LIN {X 0,Y 282.326,Z 515.053,A -85,B 0,C 180,E1 -18846.21,E2 -18846.21} C_VEL
LIN {X 0,Y 281.83,Z 513.099,A -85,B 0,C 180,E1 -18846.511,E2 -18846.511} C_VEL
LIN {X 0,Y 278.434,Z 504.389,A -85,B 0,C 180,E1 -18848.429,E2 -18848.429} C_VEL
LIN {X 0,Y 275.799,Z 498.647,A -85,B 0,C 180,E1 -18850.051,E2 -18850.051} C_VEL
LIN {X 0,Y 272.892,Z 492.622,A -85,B 0,C 180,E1 -18852.108,E2 -18852.108} C_VEL
LIN {X 0,Y 269.449,Z 485.759,A -85,B 0,C 180,E1 -18855.232,E2 -18855.232} C_VEL
LIN {X 0,Y 266.756,Z 480.992,A -85,B 0,C 180,E1 -18859.021,E2 -18859.021} C_VEL
LIN {X 0,Y 265.964,Z 478.887,A -85,B 0,C 180,E1 -18861.776,E2 -18861.776} C_VEL
LIN {X 0,Y 265.924,Z 478.099,A -85,B 0,C 180,E1 -18863.476,E2 -18863.476} C_VEL
LIN {X 0,Y 267.159,Z 478.377,A -85,B 0,C 180,E1 -18867.333,E2 -18867.333} C_VEL
LIN {X 0,Y 268.305,Z 478.984,A -85,B 0,C 180,E1 -18868.98,E2 -18868.98} C_VEL
LIN {X 0,Y 271.621,Z 482.626,A -85,B 0,C 180,E1 -18872.425,E2 -18872.425} C_VEL
LIN {X 0,Y 274.885,Z 486.681,A -85,B 0,C 180,E1 -18874.84,E2 -18874.84} C_VEL
LIN {X 0,Y 277.888,Z 490.776,A -85,B 0,C 180,E1 -18876.655,E2 -18876.655} C_VEL
LIN {X 0,Y 281.533,Z 496.331,A -85,B 0,C 180,E1 -18878.583,E2 -18878.583} C_VEL
LIN {X 0,Y 285.637,Z 503.762,A -85,B 0,C 180,E1 -18880.525,E2 -18880.525} C_VEL
LIN {X 0,Y 286.557,Z 505.613,A -85,B 0,C 180,E1 -18880.936,E2 -18880.936} C_VEL
LIN {X 0,Y 280.795,Z 557.104,A -85,B 0,C 180,E1 -18882.994,E2 -18882.994} C_VEL
LIN {X 0,Y 279.087,Z 570.067,A -85,B 0,C 180,E1 -18883.788,E2 -18883.788} C_VEL
LIN {X 0,Y 276.843,Z 582.59,A -85,B 0,C 180,E1 -18884.824,E2 -18884.824} C_VEL
LIN {X 0,Y 274.127,Z 594.365,A -85,B 0,C 180,E1 -18886.092,E2 -18886.092} C_VEL
LIN {X 0,Y 270.959,Z 605.812,A -85,B 0,C 180,E1 -18887.644,E2 -18887.644} C_VEL
LIN {X 0,Y 267.715,Z 616.024,A -85,B 0,C 180,E1 -18889.411,E2 -18889.411} C_VEL
LIN {X 0,Y 264.222,Z 625.564,A -85,B 0,C 180,E1 -18891.493,E2 -18891.493} C_VEL
LIN {X 0,Y 261.46,Z 632.41,A -85,B 0,C 180,E1 -18893.362,E2 -18893.362} C_VEL
LIN {X 0,Y 258.787,Z 638.353,A -85,B 0,C 180,E1 -18895.327,E2 -18895.327} C_VEL
LIN {X 0,Y 256.164,Z 643.857,A -85,B 0,C 180,E1 -18897.641,E2 -18897.641} C_VEL
LIN {X 0,Y 253.889,Z 648.134,A -85,B 0,C 180,E1 -18900,E2 -18900} C_VEL
LIN {X 0,Y 252.583,Z 650.359,A -85,B 0,C 180,E1 -18901.594,E2 -18901.594} C_VEL
LIN {X 0,Y 251.382,Z 652.245,A -85,B 0,C 180,E1 -18903.321,E2 -18903.321} C_VEL
LIN {X 0,Y 250.422,Z 653.517,A -85,B 0,C 180,E1 -18904.83,E2 -18904.83} C_VEL
LIN {X 0,Y 249.542,Z 654.406,A -85,B 0,C 180,E1 -18906.468,E2 -18906.468} C_VEL
LIN {X 0,Y 248.726,Z 654.929,A -85,B 0,C 180,E1 -18908.517,E2 -18908.517} C_VEL
LIN {X 0,Y 247.846,Z 654.521,A -85,B 0,C 180,E1 -18911.449,E2 -18911.449} C_VEL
LIN {X 0,Y 247.554,Z 653.658,A -85,B 0,C 180,E1 -18913.127,E2 -18913.127} C_VEL
LIN {X 0,Y 247.381,Z 652.208,A -85,B 0,C 180,E1 -18914.997,E2 -18914.997} C_VEL
LIN {X 0,Y 247.276,Z 649.517,A -85,B 0,C 180,E1 -18917.363,E2 -18917.363} C_VEL
LIN {X 0,Y 247.484,Z 645.518,A -85,B 0,C 180,E1 -18919.924,E2 -18919.924} C_VEL
LIN {X 0,Y 247.988,Z 639.143,A -85,B 0,C 180,E1 -18922.934,E2 -18922.934} C_VEL
LIN {X 0,Y 248.657,Z 632.173,A -85,B 0,C 180,E1 -18925.487,E2 -18925.487} C_VEL
LIN {X 0,Y 249.458,Z 624.632,A -85,B 0,C 180,E1 -18927.701,E2 -18927.701} C_VEL
LIN {X 0,Y 250.533,Z 614.804,A -85,B 0,C 180,E1 -18930.03,E2 -18930.03} C_VEL
LIN {X 0,Y 251.705,Z 604.3,A -85,B 0,C 180,E1 -18932.04,E2 -18932.04} C_VEL
LIN {X 0,Y 252.873,Z 593.019,A -85,B 0,C 180,E1 -18933.769,E2 -18933.769} C_VEL
LIN {X 0,Y 254.011,Z 580.659,A -85,B 0,C 180,E1 -18935.28,E2 -18935.28} C_VEL
LIN {X 0,Y 255.061,Z 566.615,A -85,B 0,C 180,E1 -18936.574,E2 -18936.574} C_VEL
LIN {X 0,Y 255.819,Z 553.718,A -85,B 0,C 180,E1 -18937.433,E2 -18937.433} C_VEL
LIN {X 0,Y 256.516,Z 534.013,A -85,B 0,C 180,E1 -18938.276,E2 -18938.276} C_VEL
LIN {X 0,Y 258.671,Z 480.462,A -85,B 0,C 180,E1 -18940.334,E2 -18940.334} C_VEL
LIN {X 0,Y 249.04,Z 452.464,A -85,B 0,C 180,E1 -18942.125,E2 -18942.125} C_VEL
LIN {X 0,Y 248.985,Z 452.468,A -85,B 0,C 180,E1 -18945.116,E2 -18945.116} C_VEL
LIN {X 0,Y 249.008,Z 452.464,A -85,B 0,C 180,E1 -18947.36,E2 -18947.36} C_VEL
LIN {X 0,Y 249.024,Z 452.466,A -85,B 0,C 180,E1 -18952.206,E2 -18952.206} C_VEL
LIN {X 0,Y 249.045,Z 452.459,A -85,B 0,C 180,E1 -18955.639,E2 -18955.639} C_VEL
LIN {X 0,Y 249.004,Z 452.465,A -85,B 0,C 180,E1 -18959.466,E2 -18959.466} C_VEL
LIN {X 0,Y 249.037,Z 452.46,A -85,B 0,C 180,E1 -18963.157,E2 -18963.157} C_VEL
LIN {X 0,Y 249.06,Z 452.461,A -85,B 0,C 180,E1 -18966.73,E2 -18966.73} C_VEL
LIN {X 0,Y 249.112,Z 452.454,A -85,B 0,C 180,E1 -18970.211,E2 -18970.211} C_VEL
LIN {X 0,Y 249.244,Z 452.435,A -85,B 0,C 180,E1 -18973.621,E2 -18973.621} C_VEL
LIN {X 0,Y 249.241,Z 452.438,A -85,B 0,C 180,E1 -18978.615,E2 -18978.615} C_VEL
LIN {X 0,Y 249.419,Z 452.413,A -85,B 0,C 180,E1 -18981.9,E2 -18981.9} C_VEL
LIN {X 0,Y 249.28,Z 452.432,A -85,B 0,C 180,E1 -18985.148,E2 -18985.148} C_VEL
LIN {X 0,Y 249.673,Z 452.385,A -85,B 0,C 180,E1 -18988.386,E2 -18988.386} C_VEL
LIN {X 0,Y 249.672,Z 452.382,A -85,B 0,C 180,E1 -18991.612,E2 -18991.612} C_VEL
LIN {X 0,Y 249.446,Z 452.413,A -85,B 0,C 180,E1 -18996.47,E2 -18996.47} C_VEL
LIN {X 0,Y 249.344,Z 452.422,A -85,B 0,C 180,E1 -18999.736,E2 -18999.736} C_VEL
LIN {X 0,Y 249.184,Z 452.445,A -85,B 0,C 180,E1 -19004.704,E2 -19004.704} C_VEL
LIN {X 0,Y 249.112,Z 452.452,A -85,B 0,C 180,E1 -19008.079,E2 -19008.079} C_VEL
LIN {X 0,Y 249.08,Z 452.456,A -85,B 0,C 180,E1 -19011.518,E2 -19011.518} C_VEL
LIN {X 0,Y 249.086,Z 452.453,A -85,B 0,C 180,E1 -19015.46,E2 -19015.46} C_VEL
LIN {X 0,Y 249.039,Z 452.463,A -85,B 0,C 180,E1 -19018.974,E2 -19018.974} C_VEL
LIN {X 0,Y 249.026,Z 452.466,A -85,B 0,C 180,E1 -19022.426,E2 -19022.426} C_VEL
LIN {X 0,Y 249.046,Z 452.462,A -85,B 0,C 180,E1 -19026.342,E2 -19026.342} C_VEL
LIN {X 0,Y 248.983,Z 452.472,A -85,B 0,C 180,E1 -19030.482,E2 -19030.482} C_VEL
LIN {X 0,Y 248.993,Z 452.468,A -85,B 0,C 180,E1 -19032.788,E2 -19032.788} C_VEL
LIN {X 0,Y 249.008,Z 452.465,A -85,B 0,C 180,E1 -19037.361,E2 -19037.361} C_VEL
LIN {X 0,Y 249.024,Z 452.46,A -85,B 0,C 180,E1 -19041.619,E2 -19041.619} C_VEL
LIN {X 0,Y 249.042,Z 452.461,A -85,B 0,C 180,E1 -19045.639,E2 -19045.639} C_VEL
LIN {X 0,Y 249.046,Z 452.458,A -85,B 0,C 180,E1 -19049.472,E2 -19049.472} C_VEL
LIN {X 0,Y 249.071,Z 452.458,A -85,B 0,C 180,E1 -19053.162,E2 -19053.162} C_VEL
LIN {X 0,Y 249.079,Z 452.458,A -85,B 0,C 180,E1 -19056.733,E2 -19056.733} C_VEL
LIN {X 0,Y 249.11,Z 452.452,A -85,B 0,C 180,E1 -19060.212,E2 -19060.212} C_VEL
LIN {X 0,Y 249.241,Z 452.436,A -85,B 0,C 180,E1 -19063.622,E2 -19063.622} C_VEL
LIN {X 0,Y 249.252,Z 452.436,A -85,B 0,C 180,E1 -19068.617,E2 -19068.617} C_VEL
LIN {X 0,Y 249.477,Z 452.407,A -85,B 0,C 180,E1 -19071.903,E2 -19071.903} C_VEL
LIN {X 0,Y 249.433,Z 452.414,A -85,B 0,C 180,E1 -19076.77,E2 -19076.77} C_VEL
LIN {X 0,Y 249.727,Z 452.376,A -85,B 0,C 180,E1 -19080,E2 -19080} C_VEL
LIN {X 0,Y 249.435,Z 452.411,A -85,B 0,C 180,E1 -19083.231,E2 -19083.231} C_VEL
LIN {X 0,Y 249.484,Z 452.406,A -85,B 0,C 180,E1 -19088.097,E2 -19088.097} C_VEL
LIN {X 0,Y 249.253,Z 452.434,A -85,B 0,C 180,E1 -19091.384,E2 -19091.384} C_VEL
LIN {X 0,Y 249.241,Z 452.437,A -85,B 0,C 180,E1 -19096.378,E2 -19096.378} C_VEL
LIN {X 0,Y 249.083,Z 452.454,A -85,B 0,C 180,E1 -19101.519,E2 -19101.519} C_VEL
LIN {X 0,Y 249.117,Z 452.452,A -85,B 0,C 180,E1 -19105.476,E2 -19105.476} C_VEL
LIN {X 0,Y 249.083,Z 452.457,A -85,B 0,C 180,E1 -19108.994,E2 -19108.994} C_VEL
LIN {X 0,Y 249.03,Z 452.462,A -85,B 0,C 180,E1 -19112.426,E2 -19112.426} C_VEL
LIN {X 0,Y 249.039,Z 452.462,A -85,B 0,C 180,E1 -19114.761,E2 -19114.761} C_VEL
LIN {X 0,Y 248.388,Z 452.546,A -85,B 0,C 180,E1 -19116.111,E2 -19116.111} C_VEL
LIN {X 0,Y 245.555,Z 452.903,A -85,B 0,C 180,E1 -19118.312,E2 -19118.312} C_VEL
LIN {X 0,Y 243.118,Z 453.205,A -85,B 0,C 180,E1 -19120.104,E2 -19120.104} C_VEL
LIN {X 0,Y 242.04,Z 453.334,A -85,B 0,C 180,E1 -19121.494,E2 -19121.494} C_VEL
LIN {X 0,Y 241.936,Z 453.345,A -85,B 0,C 180,E1 -19121.966,E2 -19121.966} C_VEL
LIN {X 0,Y 241.936,Z 453.349,A -85,B 0,C 180,E1 -19126.571,E2 -19126.571} C_VEL
LIN {X 0,Y 241.956,Z 453.343,A -85,B 0,C 180,E1 -19130.282,E2 -19130.282} C_VEL
LIN {X 0,Y 242.063,Z 453.369,A -85,B 0,C 180,E1 -19133.471,E2 -19133.471} C_VEL
LIN {X 0,Y 244.715,Z 466.337,A -85,B 0,C 180,E1 -19137.907,E2 -19137.907} C_VEL
LIN {X 0,Y 246.665,Z 475.875,A -85,B 0,C 180,E1 -19141.03,E2 -19141.03} C_VEL
LIN {X 0,Y 246.306,Z 479.6,A -85,B 0,C 180,E1 -19142.144,E2 -19142.144} C_VEL
LIN {X 0,Y 248.483,Z 510.094,A -85,B 0,C 180,E1 -19143.6,E2 -19143.6} C_VEL
LIN {X 0,Y 250.829,Z 535.634,A -85,B 0,C 180,E1 -19144.809,E2 -19144.809} C_VEL
LIN {X 0,Y 248.607,Z 589.384,A -85,B 0,C 180,E1 -19147.017,E2 -19147.017} C_VEL
LIN {X 0,Y 247.623,Z 603.29,A -85,B 0,C 180,E1 -19147.911,E2 -19147.911} C_VEL
LIN {X 0,Y 246.363,Z 616.413,A -85,B 0,C 180,E1 -19149.11,E2 -19149.11} C_VEL
LIN {X 0,Y 245.144,Z 628.254,A -85,B 0,C 180,E1 -19150.533,E2 -19150.533} C_VEL
LIN {X 0,Y 243.955,Z 638.928,A -85,B 0,C 180,E1 -19152.149,E2 -19152.149} C_VEL
LIN {X 0,Y 242.763,Z 648.961,A -85,B 0,C 180,E1 -19154.037,E2 -19154.037} C_VEL
LIN {X 0,Y 241.855,Z 658.034,A -85,B 0,C 180,E1 -19156.13,E2 -19156.13} C_VEL
LIN {X 0,Y 241.155,Z 665.499,A -85,B 0,C 180,E1 -19158.23,E2 -19158.23} C_VEL
LIN {X 0,Y 240.709,Z 672.776,A -85,B 0,C 180,E1 -19160.76,E2 -19160.76} C_VEL
LIN {X 0,Y 240.581,Z 678.564,A -85,B 0,C 180,E1 -19163.332,E2 -19163.332} C_VEL
LIN {X 0,Y 240.581,Z 682.853,A -85,B 0,C 180,E1 -19165.812,E2 -19165.812} C_VEL
LIN {X 0,Y 240.687,Z 686.021,A -85,B 0,C 180,E1 -19168.327,E2 -19168.327} C_VEL
LIN {X 0,Y 240.697,Z 687.509,A -85,B 0,C 180,E1 -19170.001,E2 -19170.001} C_VEL
LIN {X 0,Y 240.551,Z 688.525,A -85,B 0,C 180,E1 -19171.675,E2 -19171.675} C_VEL
LIN {X 0,Y 240.183,Z 689.037,A -85,B 0,C 180,E1 -19173.356,E2 -19173.356} C_VEL
LIN {X 0,Y 240.093,Z 689.117,A -85,B 0,C 180,E1 -19175.586,E2 -19175.586} C_VEL
LIN {X 0,Y 240.16,Z 688.153,A -85,B 0,C 180,E1 -19178.414,E2 -19178.414} C_VEL
LIN {X 0,Y 240.473,Z 687.031,A -85,B 0,C 180,E1 -19180.1,E2 -19180.1} C_VEL
LIN {X 0,Y 241.585,Z 683.542,A -85,B 0,C 180,E1 -19183.458,E2 -19183.458} C_VEL
LIN {X 0,Y 243.176,Z 679.816,A -85,B 0,C 180,E1 -19185.936,E2 -19185.936} C_VEL
LIN {X 0,Y 245.077,Z 675.065,A -85,B 0,C 180,E1 -19188.388,E2 -19188.388} C_VEL
LIN {X 0,Y 248.042,Z 668.056,A -85,B 0,C 180,E1 -19191.178,E2 -19191.178} C_VEL
LIN {X 0,Y 251.761,Z 659.198,A -85,B 0,C 180,E1 -19193.878,E2 -19193.878} C_VEL
LIN {X 0,Y 255.594,Z 649.847,A -85,B 0,C 180,E1 -19196.101,E2 -19196.101} C_VEL
LIN {X 0,Y 259.509,Z 639.305,A -85,B 0,C 180,E1 -19198.071,E2 -19198.071} C_VEL
LIN {X 0,Y 263.479,Z 627.709,A -85,B 0,C 180,E1 -19199.789,E2 -19199.789} C_VEL
LIN {X 0,Y 267.052,Z 616.215,A -85,B 0,C 180,E1 -19201.097,E2 -19201.097} C_VEL
LIN {X 0,Y 270.567,Z 602.674,A -85,B 0,C 180,E1 -19202.284,E2 -19202.284} C_VEL
LIN {X 0,Y 273.295,Z 589,A -85,B 0,C 180,E1 -19203.18,E2 -19203.18} C_VEL
LIN {X 0,Y 275.538,Z 574.021,A -85,B 0,C 180,E1 -19203.86,E2 -19203.86} C_VEL
LIN {X 0,Y 279.213,Z 541.099,A -85,B 0,C 180,E1 -19205.196,E2 -19205.196} C_VEL
LIN {X 0,Y 279.022,Z 528.795,A -85,B 0,C 180,E1 -19206.177,E2 -19206.177} C_VEL
LIN {X 0,Y 278.4,Z 518.134,A -85,B 0,C 180,E1 -19207.26,E2 -19207.26} C_VEL
LIN {X 0,Y 275.283,Z 509.663,A -85,B 0,C 180,E1 -19209.169,E2 -19209.169} C_VEL
LIN {X 0,Y 272.972,Z 504.355,A -85,B 0,C 180,E1 -19210.707,E2 -19210.707} C_VEL
LIN {X 0,Y 270.596,Z 498.97,A -85,B 0,C 180,E1 -19212.564,E2 -19212.564} C_VEL
LIN {X 0,Y 267.41,Z 492.248,A -85,B 0,C 180,E1 -19215.677,E2 -19215.677} C_VEL
LIN {X 0,Y 265.082,Z 487.715,A -85,B 0,C 180,E1 -19219.345,E2 -19219.345} C_VEL
LIN {X 0,Y 264.402,Z 485.554,A -85,B 0,C 180,E1 -19222.312,E2 -19222.312} C_VEL
LIN {X 0,Y 264.526,Z 484.953,A -85,B 0,C 180,E1 -19224.232,E2 -19224.232} C_VEL
LIN {X 0,Y 266.105,Z 485.466,A -85,B 0,C 180,E1 -19228.115,E2 -19228.115} C_VEL
LIN {X 0,Y 266.971,Z 486.316,A -85,B 0,C 180,E1 -19229.286,E2 -19229.286} C_VEL
LIN {X 0,Y 269.719,Z 489.366,A -85,B 0,C 180,E1 -19232.161,E2 -19232.161} C_VEL
LIN {X 0,Y 272.655,Z 493.167,A -85,B 0,C 180,E1 -19234.446,E2 -19234.446} C_VEL
LIN {X 0,Y 275.309,Z 497.029,A -85,B 0,C 180,E1 -19236.173,E2 -19236.173} C_VEL
LIN {X 0,Y 278.098,Z 501.457,A -85,B 0,C 180,E1 -19237.779,E2 -19237.779} C_VEL
LIN {X 0,Y 281.912,Z 508.483,A -85,B 0,C 180,E1 -19239.743,E2 -19239.743} C_VEL
LIN {X 0,Y 282.164,Z 509.341,A -85,B 0,C 180,E1 -19239.89,E2 -19239.89} C_VEL
LIN {X 0,Y 276.44,Z 557.647,A -85,B 0,C 180,E1 -19241.843,E2 -19241.843} C_VEL
LIN {X 0,Y 274.71,Z 570.009,A -85,B 0,C 180,E1 -19242.61,E2 -19242.61} C_VEL
LIN {X 0,Y 272.153,Z 583.297,A -85,B 0,C 180,E1 -19243.709,E2 -19243.709} C_VEL
LIN {X 0,Y 269.12,Z 595.783,A -85,B 0,C 180,E1 -19245.074,E2 -19245.074} C_VEL
LIN {X 0,Y 265.798,Z 606.936,A -85,B 0,C 180,E1 -19246.623,E2 -19246.623} C_VEL
LIN {X 0,Y 262.351,Z 616.95,A -85,B 0,C 180,E1 -19248.409,E2 -19248.409} C_VEL
LIN {X 0,Y 258.505,Z 626.84,A -85,B 0,C 180,E1 -19250.612,E2 -19250.612} C_VEL
LIN {X 0,Y 255.264,Z 634.243,A -85,B 0,C 180,E1 -19252.723,E2 -19252.723} C_VEL
LIN {X 0,Y 251.834,Z 641.075,A -85,B 0,C 180,E1 -19255.197,E2 -19255.197} C_VEL
LIN {X 0,Y 249.126,Z 646.135,A -85,B 0,C 180,E1 -19257.575,E2 -19257.575} C_VEL
LIN {X 0,Y 246.789,Z 650.03,A -85,B 0,C 180,E1 -19260,E2 -19260} C_VEL
LIN {X 0,Y 245.477,Z 652.035,A -85,B 0,C 180,E1 -19261.64,E2 -19261.64} C_VEL
LIN {X 0,Y 244.309,Z 653.549,A -85,B 0,C 180,E1 -19263.298,E2 -19263.298} C_VEL
LIN {X 0,Y 243.262,Z 654.657,A -85,B 0,C 180,E1 -19264.972,E2 -19264.972} C_VEL
LIN {X 0,Y 242.391,Z 655.359,A -85,B 0,C 180,E1 -19266.66,E2 -19266.66} C_VEL
LIN {X 0,Y 241.641,Z 655.588,A -85,B 0,C 180,E1 -19268.551,E2 -19268.551} C_VEL
LIN {X 0,Y 240.696,Z 654.78,A -85,B 0,C 180,E1 -19271.794,E2 -19271.794} C_VEL
LIN {X 0,Y 240.436,Z 653.716,A -85,B 0,C 180,E1 -19273.523,E2 -19273.523} C_VEL
LIN {X 0,Y 240.233,Z 651.242,A -85,B 0,C 180,E1 -19276.136,E2 -19276.136} C_VEL
LIN {X 0,Y 240.279,Z 647.625,A -85,B 0,C 180,E1 -19278.768,E2 -19278.768} C_VEL
LIN {X 0,Y 240.591,Z 642.722,A -85,B 0,C 180,E1 -19281.431,E2 -19281.431} C_VEL
LIN {X 0,Y 241.136,Z 636.448,A -85,B 0,C 180,E1 -19284.081,E2 -19284.081} C_VEL
LIN {X 0,Y 241.975,Z 628.435,A -85,B 0,C 180,E1 -19286.756,E2 -19286.756} C_VEL
LIN {X 0,Y 242.889,Z 620.108,A -85,B 0,C 180,E1 -19288.99,E2 -19288.99} C_VEL
LIN {X 0,Y 244.039,Z 609.913,A -85,B 0,C 180,E1 -19291.223,E2 -19291.223} C_VEL
LIN {X 0,Y 245.209,Z 598.821,A -85,B 0,C 180,E1 -19293.167,E2 -19293.167} C_VEL
LIN {X 0,Y 246.406,Z 587.366,A -85,B 0,C 180,E1 -19294.781,E2 -19294.781} C_VEL
LIN {X 0,Y 247.459,Z 575.374,A -85,B 0,C 180,E1 -19296.108,E2 -19296.108} C_VEL
LIN {X 0,Y 248.529,Z 560.848,A -85,B 0,C 180,E1 -19297.308,E2 -19297.308} C_VEL
LIN {X 0,Y 249.158,Z 547.242,A -85,B 0,C 180,E1 -19298.074,E2 -19298.074} C_VEL
LIN {X 0,Y 251.767,Z 481.763,A -85,B 0,C 180,E1 -19300.686,E2 -19300.686} C_VEL
LIN {X 0,Y 241.975,Z 453.345,A -85,B 0,C 180,E1 -19302.592,E2 -19302.592} C_VEL
LIN {X 0,Y 241.924,Z 453.35,A -85,B 0,C 180,E1 -19306.574,E2 -19306.574} C_VEL
LIN {X 0,Y 241.938,Z 453.349,A -85,B 0,C 180,E1 -19310.276,E2 -19310.276} C_VEL
LIN {X 0,Y 241.975,Z 453.343,A -85,B 0,C 180,E1 -19314.486,E2 -19314.486} C_VEL
LIN {X 0,Y 241.955,Z 453.348,A -85,B 0,C 180,E1 -19318.476,E2 -19318.476} C_VEL
LIN {X 0,Y 241.97,Z 453.344,A -85,B 0,C 180,E1 -19322.307,E2 -19322.307} C_VEL
LIN {X 0,Y 242.029,Z 453.336,A -85,B 0,C 180,E1 -19326.012,E2 -19326.012} C_VEL
LIN {X 0,Y 242.039,Z 453.333,A -85,B 0,C 180,E1 -19329.607,E2 -19329.607} C_VEL
LIN {X 0,Y 242.165,Z 453.317,A -85,B 0,C 180,E1 -19333.278,E2 -19333.278} C_VEL
LIN {X 0,Y 242.178,Z 453.319,A -85,B 0,C 180,E1 -19338.279,E2 -19338.279} C_VEL
LIN {X 0,Y 242.373,Z 453.29,A -85,B 0,C 180,E1 -19341.663,E2 -19341.663} C_VEL
LIN {X 0,Y 242.24,Z 453.309,A -85,B 0,C 180,E1 -19345.006,E2 -19345.006} C_VEL
LIN {X 0,Y 242.634,Z 453.261,A -85,B 0,C 180,E1 -19348.34,E2 -19348.34} C_VEL
LIN {X 0,Y 242.632,Z 453.259,A -85,B 0,C 180,E1 -19351.659,E2 -19351.659} C_VEL
LIN {X 0,Y 242.417,Z 453.287,A -85,B 0,C 180,E1 -19356.659,E2 -19356.659} C_VEL
LIN {X 0,Y 242.268,Z 453.305,A -85,B 0,C 180,E1 -19360.023,E2 -19360.023} C_VEL
LIN {X 0,Y 242.14,Z 453.319,A -85,B 0,C 180,E1 -19365.142,E2 -19365.142} C_VEL
LIN {X 0,Y 242.05,Z 453.335,A -85,B 0,C 180,E1 -19368.625,E2 -19368.625} C_VEL
LIN {X 0,Y 242.003,Z 453.34,A -85,B 0,C 180,E1 -19372.18,E2 -19372.18} C_VEL
LIN {X 0,Y 242.032,Z 453.332,A -85,B 0,C 180,E1 -19375.82,E2 -19375.82} C_VEL
LIN {X 0,Y 241.969,Z 453.342,A -85,B 0,C 180,E1 -19379.588,E2 -19379.588} C_VEL
LIN {X 0,Y 241.978,Z 453.338,A -85,B 0,C 180,E1 -19383.492,E2 -19383.492} C_VEL
LIN {X 0,Y 241.986,Z 453.34,A -85,B 0,C 180,E1 -19387.582,E2 -19387.582} C_VEL
LIN {X 0,Y 241.922,Z 453.347,A -85,B 0,C 180,E1 -19391.925,E2 -19391.925} C_VEL
LIN {X 0,Y 241.924,Z 453.352,A -85,B 0,C 180,E1 -19396.573,E2 -19396.573} C_VEL
LIN {X 0,Y 241.955,Z 453.345,A -85,B 0,C 180,E1 -19400.281,E2 -19400.281} C_VEL
LIN {X 0,Y 241.98,Z 453.344,A -85,B 0,C 180,E1 -19404.488,E2 -19404.488} C_VEL
LIN {X 0,Y 241.972,Z 453.345,A -85,B 0,C 180,E1 -19408.48,E2 -19408.48} C_VEL
LIN {X 0,Y 242.002,Z 453.339,A -85,B 0,C 180,E1 -19412.312,E2 -19412.312} C_VEL
LIN {X 0,Y 242.057,Z 453.332,A -85,B 0,C 180,E1 -19416.016,E2 -19416.016} C_VEL
LIN {X 0,Y 242.037,Z 453.331,A -85,B 0,C 180,E1 -19419.608,E2 -19419.608} C_VEL
LIN {X 0,Y 242.162,Z 453.318,A -85,B 0,C 180,E1 -19423.278,E2 -19423.278} C_VEL
LIN {X 0,Y 242.186,Z 453.314,A -85,B 0,C 180,E1 -19428.28,E2 -19428.28} C_VEL
LIN {X 0,Y 242.424,Z 453.285,A -85,B 0,C 180,E1 -19431.666,E2 -19431.666} C_VEL
LIN {X 0,Y 242.254,Z 453.306,A -85,B 0,C 180,E1 -19435.007,E2 -19435.007} C_VEL
LIN {X 0,Y 242.635,Z 453.26,A -85,B 0,C 180,E1 -19438.34,E2 -19438.34} C_VEL
LIN {X 0,Y 242.635,Z 453.259,A -85,B 0,C 180,E1 -19441.66,E2 -19441.66} C_VEL
LIN {X 0,Y 242.433,Z 453.286,A -85,B 0,C 180,E1 -19446.659,E2 -19446.659} C_VEL
LIN {X 0,Y 242.345,Z 453.296,A -85,B 0,C 180,E1 -19450.021,E2 -19450.021} C_VEL
LIN {X 0,Y 242.166,Z 453.318,A -85,B 0,C 180,E1 -19455.141,E2 -19455.141} C_VEL
LIN {X 0,Y 242.072,Z 453.333,A -85,B 0,C 180,E1 -19458.624,E2 -19458.624} C_VEL
LIN {X 0,Y 242.006,Z 453.336,A -85,B 0,C 180,E1 -19462.181,E2 -19462.181} C_VEL
LIN {X 0,Y 242.066,Z 453.33,A -85,B 0,C 180,E1 -19465.838,E2 -19465.838} C_VEL
LIN {X 0,Y 242.03,Z 453.333,A -85,B 0,C 180,E1 -19469.58,E2 -19469.58} C_VEL
LIN {X 0,Y 241.98,Z 453.34,A -85,B 0,C 180,E1 -19473.493,E2 -19473.493} C_VEL
LIN {X 0,Y 241.989,Z 453.339,A -85,B 0,C 180,E1 -19477.582,E2 -19477.582} C_VEL
LIN {X 0,Y 241.936,Z 453.345,A -85,B 0,C 180,E1 -19481.966,E2 -19481.966} C_VEL
LIN {X 0,Y 241.227,Z 453.436,A -85,B 0,C 180,E1 -19483.355,E2 -19483.355} C_VEL
LIN {X 0,Y 238.377,Z 453.789,A -85,B 0,C 180,E1 -19485.622,E2 -19485.622} C_VEL
LIN {X 0,Y 235.981,Z 454.09,A -85,B 0,C 180,E1 -19487.469,E2 -19487.469} C_VEL
LIN {X 0,Y 234.952,Z 454.217,A -85,B 0,C 180,E1 -19488.902,E2 -19488.902} C_VEL
LIN {X 0,Y 234.866,Z 454.224,A -85,B 0,C 180,E1 -19489.387,E2 -19489.387} C_VEL
LIN {X 0,Y 235.021,Z 454.306,A -85,B 0,C 180,E1 -19493.202,E2 -19493.202} C_VEL
LIN {X 0,Y 237.71,Z 467.519,A -85,B 0,C 180,E1 -19497.848,E2 -19497.848} C_VEL
LIN {X 0,Y 239.623,Z 476.982,A -85,B 0,C 180,E1 -19501.031,E2 -19501.031} C_VEL
LIN {X 0,Y 239.401,Z 478.938,A -85,B 0,C 180,E1 -19501.65,E2 -19501.65} C_VEL
LIN {X 0,Y 241.445,Z 508.632,A -85,B 0,C 180,E1 -19503.126,E2 -19503.126} C_VEL
LIN {X 0,Y 243.914,Z 535.614,A -85,B 0,C 180,E1 -19504.45,E2 -19504.45} C_VEL
LIN {X 0,Y 241.564,Z 589.707,A -85,B 0,C 180,E1 -19506.761,E2 -19506.761} C_VEL
LIN {X 0,Y 240.599,Z 603.374,A -85,B 0,C 180,E1 -19507.683,E2 -19507.683} C_VEL
LIN {X 0,Y 239.331,Z 616.305,A -85,B 0,C 180,E1 -19508.917,E2 -19508.917} C_VEL
LIN {X 0,Y 238.099,Z 628.024,A -85,B 0,C 180,E1 -19510.382,E2 -19510.382} C_VEL
LIN {X 0,Y 236.817,Z 639.25,A -85,B 0,C 180,E1 -19512.165,E2 -19512.165} C_VEL
LIN {X 0,Y 235.693,Z 648.551,A -85,B 0,C 180,E1 -19513.99,E2 -19513.99} C_VEL
LIN {X 0,Y 234.767,Z 657.567,A -85,B 0,C 180,E1 -19516.144,E2 -19516.144} C_VEL
LIN {X 0,Y 234.078,Z 664.993,A -85,B 0,C 180,E1 -19518.308,E2 -19518.308} C_VEL
LIN {X 0,Y 233.65,Z 672.236,A -85,B 0,C 180,E1 -19520.915,E2 -19520.915} C_VEL
LIN {X 0,Y 233.519,Z 677.516,A -85,B 0,C 180,E1 -19523.302,E2 -19523.302} C_VEL
LIN {X 0,Y 233.551,Z 681.673,A -85,B 0,C 180,E1 -19525.686,E2 -19525.686} C_VEL
LIN {X 0,Y 233.639,Z 685.012,A -85,B 0,C 180,E1 -19528.277,E2 -19528.277} C_VEL
LIN {X 0,Y 233.661,Z 686.583,A -85,B 0,C 180,E1 -19530.001,E2 -19530.001} C_VEL
LIN {X 0,Y 233.487,Z 687.681,A -85,B 0,C 180,E1 -19531.726,E2 -19531.726} C_VEL
LIN {X 0,Y 233.109,Z 688.311,A -85,B 0,C 180,E1 -19533.458,E2 -19533.458} C_VEL
LIN {X 0,Y 233.03,Z 688.498,A -85,B 0,C 180,E1 -19535.582,E2 -19535.582} C_VEL
LIN {X 0,Y 233.101,Z 687.69,A -85,B 0,C 180,E1 -19538.671,E2 -19538.671} C_VEL
LIN {X 0,Y 233.448,Z 686.687,A -85,B 0,C 180,E1 -19540.407,E2 -19540.407} C_VEL
LIN {X 0,Y 233.913,Z 685.281,A -85,B 0,C 180,E1 -19542.142,E2 -19542.142} C_VEL
LIN {X 0,Y 235.2,Z 682.394,A -85,B 0,C 180,E1 -19544.714,E2 -19544.714} C_VEL
LIN {X 0,Y 236.922,Z 678.523,A -85,B 0,C 180,E1 -19547.256,E2 -19547.256} C_VEL
LIN {X 0,Y 239.729,Z 672.449,A -85,B 0,C 180,E1 -19550.26,E2 -19550.26} C_VEL
LIN {X 0,Y 243.075,Z 665.266,A -85,B 0,C 180,E1 -19552.975,E2 -19552.975} C_VEL
LIN {X 0,Y 246.648,Z 657.384,A -85,B 0,C 180,E1 -19555.304,E2 -19555.304} C_VEL
LIN {X 0,Y 250.781,Z 647.803,A -85,B 0,C 180,E1 -19557.543,E2 -19557.543} C_VEL
LIN {X 0,Y 254.987,Z 637.136,A -85,B 0,C 180,E1 -19559.517,E2 -19559.517} C_VEL
LIN {X 0,Y 258.839,Z 626.51,A -85,B 0,C 180,E1 -19561.058,E2 -19561.058} C_VEL
LIN {X 0,Y 262.608,Z 614.873,A -85,B 0,C 180,E1 -19562.361,E2 -19562.361} C_VEL
LIN {X 0,Y 266.302,Z 601.416,A -85,B 0,C 180,E1 -19563.544,E2 -19563.544} C_VEL
LIN {X 0,Y 269.043,Z 588.511,A -85,B 0,C 180,E1 -19564.396,E2 -19564.396} C_VEL
LIN {X 0,Y 271.392,Z 573.761,A -85,B 0,C 180,E1 -19565.074,E2 -19565.074} C_VEL
LIN {X 0,Y 275.078,Z 542.504,A -85,B 0,C 180,E1 -19566.353,E2 -19566.353} C_VEL
LIN {X 0,Y 275.116,Z 531.447,A -85,B 0,C 180,E1 -19567.272,E2 -19567.272} C_VEL
LIN {X 0,Y 274.738,Z 522.333,A -85,B 0,C 180,E1 -19568.2,E2 -19568.2} C_VEL
LIN {X 0,Y 272.158,Z 514.807,A -85,B 0,C 180,E1 -19569.983,E2 -19569.983} C_VEL
LIN {X 0,Y 270.216,Z 510.059,A -85,B 0,C 180,E1 -19571.4,E2 -19571.4} C_VEL
LIN {X 0,Y 268.024,Z 504.852,A -85,B 0,C 180,E1 -19573.252,E2 -19573.252} C_VEL
LIN {X 0,Y 265.419,Z 498.75,A -85,B 0,C 180,E1 -19576.138,E2 -19576.138} C_VEL
LIN {X 0,Y 263.452,Z 494.549,A -85,B 0,C 180,E1 -19579.551,E2 -19579.551} C_VEL
LIN {X 0,Y 262.874,Z 492.459,A -85,B 0,C 180,E1 -19582.393,E2 -19582.393} C_VEL
LIN {X 0,Y 262.96,Z 491.928,A -85,B 0,C 180,E1 -19583.986,E2 -19583.986} C_VEL
LIN {X 0,Y 263.953,Z 492.179,A -85,B 0,C 180,E1 -19587.045,E2 -19587.045} C_VEL
LIN {X 0,Y 265.012,Z 492.824,A -85,B 0,C 180,E1 -19588.738,E2 -19588.738} C_VEL
LIN {X 0,Y 267.72,Z 495.989,A -85,B 0,C 180,E1 -19591.802,E2 -19591.802} C_VEL
LIN {X 0,Y 270.454,Z 499.702,A -85,B 0,C 180,E1 -19594.067,E2 -19594.067} C_VEL
LIN {X 0,Y 272.924,Z 503.464,A -85,B 0,C 180,E1 -19595.782,E2 -19595.782} C_VEL
LIN {X 0,Y 275.686,Z 508.112,A -85,B 0,C 180,E1 -19597.464,E2 -19597.464} C_VEL
LIN {X 0,Y 278.059,Z 512.857,A -85,B 0,C 180,E1 -19598.773,E2 -19598.773} C_VEL
LIN {X 0,Y 272.124,Z 559.655,A -85,B 0,C 180,E1 -19600.725,E2 -19600.725} C_VEL
LIN {X 0,Y 269.994,Z 573.18,A -85,B 0,C 180,E1 -19601.602,E2 -19601.602} C_VEL
LIN {X 0,Y 267.554,Z 584.854,A -85,B 0,C 180,E1 -19602.615,E2 -19602.615} C_VEL
LIN {X 0,Y 264.289,Z 597.102,A -85,B 0,C 180,E1 -19603.996,E2 -19603.996} C_VEL
LIN {X 0,Y 260.4,Z 609.115,A -85,B 0,C 180,E1 -19605.723,E2 -19605.723} C_VEL
LIN {X 0,Y 256.407,Z 619.89,A -85,B 0,C 180,E1 -19607.735,E2 -19607.735} C_VEL
LIN {X 0,Y 252.347,Z 629.215,A -85,B 0,C 180,E1 -19609.976,E2 -19609.976} C_VEL
LIN {X 0,Y 248.773,Z 636.644,A -85,B 0,C 180,E1 -19612.245,E2 -19612.245} C_VEL
LIN {X 0,Y 245.92,Z 641.937,A -85,B 0,C 180,E1 -19614.259,E2 -19614.259} C_VEL
LIN {X 0,Y 242.959,Z 646.935,A -85,B 0,C 180,E1 -19616.683,E2 -19616.683} C_VEL
LIN {X 0,Y 240.437,Z 650.766,A -85,B 0,C 180,E1 -19619.162,E2 -19619.162} C_VEL
LIN {X 0,Y 238.33,Z 653.561,A -85,B 0,C 180,E1 -19621.69,E2 -19621.69} C_VEL
LIN {X 0,Y 237.136,Z 654.883,A -85,B 0,C 180,E1 -19623.398,E2 -19623.398} C_VEL
LIN {X 0,Y 236.088,Z 655.736,A -85,B 0,C 180,E1 -19625.124,E2 -19625.124} C_VEL
LIN {X 0,Y 235.208,Z 656.173,A -85,B 0,C 180,E1 -19626.864,E2 -19626.864} C_VEL
LIN {X 0,Y 234.53,Z 656.201,A -85,B 0,C 180,E1 -19628.617,E2 -19628.617} C_VEL
LIN {X 0,Y 233.94,Z 655.788,A -85,B 0,C 180,E1 -19630.384,E2 -19630.384} C_VEL
LIN {X 0,Y 233.528,Z 654.913,A -85,B 0,C 180,E1 -19632.161,E2 -19632.161} C_VEL
LIN {X 0,Y 233.17,Z 652.311,A -85,B 0,C 180,E1 -19635.306,E2 -19635.306} C_VEL
LIN {X 0,Y 233.153,Z 648.237,A -85,B 0,C 180,E1 -19638.452,E2 -19638.452} C_VEL
LIN {X 0,Y 233.472,Z 643.397,A -85,B 0,C 180,E1 -19641.175,E2 -19641.175} C_VEL
LIN {X 0,Y 234.015,Z 637.104,A -85,B 0,C 180,E1 -19643.918,E2 -19643.918} C_VEL
LIN {X 0,Y 234.705,Z 630.438,A -85,B 0,C 180,E1 -19646.254,E2 -19646.254} C_VEL
LIN {X 0,Y 235.555,Z 622.604,A -85,B 0,C 180,E1 -19648.514,E2 -19648.514} C_VEL
LIN {X 0,Y 236.782,Z 611.806,A -85,B 0,C 180,E1 -19651.019,E2 -19651.019} C_VEL
LIN {X 0,Y 237.879,Z 601.916,A -85,B 0,C 180,E1 -19652.88,E2 -19652.88} C_VEL
LIN {X 0,Y 239.138,Z 590.416,A -85,B 0,C 180,E1 -19654.624,E2 -19654.624} C_VEL
LIN {X 0,Y 240.325,Z 577.384,A -85,B 0,C 180,E1 -19656.182,E2 -19656.182} C_VEL
LIN {X 0,Y 241.29,Z 564.815,A -85,B 0,C 180,E1 -19657.315,E2 -19657.315} C_VEL
LIN {X 0,Y 241.997,Z 551.051,A -85,B 0,C 180,E1 -19658.214,E2 -19658.214} C_VEL
LIN {X 0,Y 244.871,Z 483.139,A -85,B 0,C 180,E1 -19661.055,E2 -19661.055} C_VEL
LIN {X 0,Y 234.959,Z 454.501,A -85,B 0,C 180,E1 -19662.985,E2 -19662.985} C_VEL
LIN {X 0,Y 234.897,Z 454.224,A -85,B 0,C 180,E1 -19663.179,E2 -19663.179} C_VEL
LIN {X 0,Y 234.877,Z 454.228,A -85,B 0,C 180,E1 -19666.511,E2 -19666.511} C_VEL
LIN {X 0,Y 234.919,Z 454.22,A -85,B 0,C 180,E1 -19671.078,E2 -19671.078} C_VEL
LIN {X 0,Y 234.924,Z 454.218,A -85,B 0,C 180,E1 -19675.36,E2 -19675.36} C_VEL
LIN {X 0,Y 234.901,Z 454.222,A -85,B 0,C 180,E1 -19679.427,E2 -19679.427} C_VEL
LIN {X 0,Y 234.97,Z 454.212,A -85,B 0,C 180,E1 -19683.806,E2 -19683.806} C_VEL
LIN {X 0,Y 235.001,Z 454.21,A -85,B 0,C 180,E1 -19688.968,E2 -19688.968} C_VEL
LIN {X 0,Y 235.099,Z 454.197,A -85,B 0,C 180,E1 -19693.059,E2 -19693.059} C_VEL
LIN {X 0,Y 235.112,Z 454.197,A -85,B 0,C 180,E1 -19697.921,E2 -19697.921} C_VEL
LIN {X 0,Y 235.313,Z 454.169,A -85,B 0,C 180,E1 -19701.411,E2 -19701.411} C_VEL
LIN {X 0,Y 235.351,Z 454.167,A -85,B 0,C 180,E1 -19703.139,E2 -19703.139} C_VEL
LIN {X 0,Y 235.593,Z 454.138,A -85,B 0,C 180,E1 -19708.29,E2 -19708.29} C_VEL
LIN {X 0,Y 235.591,Z 454.136,A -85,B 0,C 180,E1 -19711.709,E2 -19711.709} C_VEL
LIN {X 0,Y 235.367,Z 454.163,A -85,B 0,C 180,E1 -19716.859,E2 -19716.859} C_VEL
LIN {X 0,Y 235.215,Z 454.185,A -85,B 0,C 180,E1 -19720.327,E2 -19720.327} C_VEL
LIN {X 0,Y 235.086,Z 454.197,A -85,B 0,C 180,E1 -19725.608,E2 -19725.608} C_VEL
LIN {X 0,Y 234.99,Z 454.212,A -85,B 0,C 180,E1 -19729.207,E2 -19729.207} C_VEL
LIN {X 0,Y 234.946,Z 454.217,A -85,B 0,C 180,E1 -19732.884,E2 -19732.884} C_VEL
LIN {X 0,Y 234.945,Z 454.22,A -85,B 0,C 180,E1 -19736.66,E2 -19736.66} C_VEL
LIN {X 0,Y 234.898,Z 454.226,A -85,B 0,C 180,E1 -19740.572,E2 -19740.572} C_VEL
LIN {X 0,Y 234.929,Z 454.22,A -85,B 0,C 180,E1 -19744.638,E2 -19744.638} C_VEL
LIN {X 0,Y 234.91,Z 454.223,A -85,B 0,C 180,E1 -19748.935,E2 -19748.935} C_VEL
LIN {X 0,Y 234.873,Z 454.224,A -85,B 0,C 180,E1 -19753.489,E2 -19753.489} C_VEL
LIN {X 0,Y 234.877,Z 454.229,A -85,B 0,C 180,E1 -19756.512,E2 -19756.512} C_VEL
LIN {X 0,Y 234.917,Z 454.218,A -85,B 0,C 180,E1 -19761.078,E2 -19761.078} C_VEL
LIN {X 0,Y 234.926,Z 454.22,A -85,B 0,C 180,E1 -19765.361,E2 -19765.361} C_VEL
LIN {X 0,Y 234.921,Z 454.217,A -85,B 0,C 180,E1 -19769.431,E2 -19769.431} C_VEL
LIN {X 0,Y 234.993,Z 454.211,A -85,B 0,C 180,E1 -19773.794,E2 -19773.794} C_VEL
LIN {X 0,Y 235.011,Z 454.208,A -85,B 0,C 180,E1 -19778.97,E2 -19778.97} C_VEL
LIN {X 0,Y 235.096,Z 454.2,A -85,B 0,C 180,E1 -19783.059,E2 -19783.059} C_VEL
LIN {X 0,Y 235.118,Z 454.192,A -85,B 0,C 180,E1 -19787.922,E2 -19787.922} C_VEL
LIN {X 0,Y 235.374,Z 454.164,A -85,B 0,C 180,E1 -19791.414,E2 -19791.414} C_VEL
LIN {X 0,Y 235.4,Z 454.161,A -85,B 0,C 180,E1 -19793.141,E2 -19793.141} C_VEL
LIN {X 0,Y 235.594,Z 454.136,A -85,B 0,C 180,E1 -19798.291,E2 -19798.291} C_VEL
LIN {X 0,Y 235.595,Z 454.136,A -85,B 0,C 180,E1 -19801.71,E2 -19801.71} C_VEL
LIN {X 0,Y 235.405,Z 454.162,A -85,B 0,C 180,E1 -19806.859,E2 -19806.859} C_VEL
LIN {X 0,Y 235.253,Z 454.181,A -85,B 0,C 180,E1 -19810.326,E2 -19810.326} C_VEL
LIN {X 0,Y 235.113,Z 454.195,A -85,B 0,C 180,E1 -19815.607,E2 -19815.607} C_VEL
LIN {X 0,Y 235.007,Z 454.21,A -85,B 0,C 180,E1 -19819.206,E2 -19819.206} C_VEL
LIN {X 0,Y 234.952,Z 454.217,A -85,B 0,C 180,E1 -19822.884,E2 -19822.884} C_VEL
LIN {X 0,Y 234.969,Z 454.218,A -85,B 0,C 180,E1 -19826.658,E2 -19826.658} C_VEL
LIN {X 0,Y 234.931,Z 454.22,A -85,B 0,C 180,E1 -19830.568,E2 -19830.568} C_VEL
LIN {X 0,Y 234.93,Z 454.222,A -85,B 0,C 180,E1 -19834.638,E2 -19834.638} C_VEL
LIN {X 0,Y 234.941,Z 454.217,A -85,B 0,C 180,E1 -19838.945,E2 -19838.945} C_VEL
LIN {X 0,Y 234.89,Z 454.224,A -85,B 0,C 180,E1 -19843.486,E2 -19843.486} C_VEL
LIN {X 0,Y 234.889,Z 454.226,A -85,B 0,C 180,E1 -19846.515,E2 -19846.515} C_VEL
LIN {X 0,Y 234.866,Z 454.224,A -85,B 0,C 180,E1 -19849.387,E2 -19849.387} C_VEL
LIN {X 0,Y 234.206,Z 454.323,A -85,B 0,C 180,E1 -19850.371,E2 -19850.371} C_VEL
LIN {X 0,Y 231.52,Z 455.083,A -85,B 0,C 180,E1 -19851.924,E2 -19851.924} C_VEL
LIN {X 0,Y 229.425,Z 456.503,A -85,B 0,C 180,E1 -19853.126,E2 -19853.126} C_VEL
LIN {X 0,Y 228.696,Z 458.397,A -85,B 0,C 180,E1 -19854.085,E2 -19854.085} C_VEL
LIN {X 0,Y 228.747,Z 458.941,A -85,B 0,C 180,E1 -19854.295,E2 -19854.295} C_VEL
LIN {X 0,Y 231.676,Z 473.47,A -85,B 0,C 180,E1 -19859.462,E2 -19859.462} C_VEL
LIN {X 0,Y 232.49,Z 478.479,A -85,B 0,C 180,E1 -19861.175,E2 -19861.175} C_VEL
LIN {X 0,Y 234.348,Z 506.669,A -85,B 0,C 180,E1 -19862.605,E2 -19862.605} C_VEL
LIN {X 0,Y 236.938,Z 536.82,A -85,B 0,C 180,E1 -19864.137,E2 -19864.137} C_VEL
LIN {X 0,Y 234.63,Z 588.647,A -85,B 0,C 180,E1 -19866.442,E2 -19866.442} C_VEL
LIN {X 0,Y 233.724,Z 601.702,A -85,B 0,C 180,E1 -19867.34,E2 -19867.34} C_VEL
LIN {X 0,Y 232.492,Z 613.933,A -85,B 0,C 180,E1 -19868.499,E2 -19868.499} C_VEL
LIN {X 0,Y 231.198,Z 625.958,A -85,B 0,C 180,E1 -19870.003,E2 -19870.003} C_VEL
LIN {X 0,Y 229.97,Z 636.78,A -85,B 0,C 180,E1 -19871.708,E2 -19871.708} C_VEL
LIN {X 0,Y 228.866,Z 646.038,A -85,B 0,C 180,E1 -19873.499,E2 -19873.499} C_VEL
LIN {X 0,Y 227.868,Z 655.378,A -85,B 0,C 180,E1 -19875.716,E2 -19875.716} C_VEL
LIN {X 0,Y 227.144,Z 663.077,A -85,B 0,C 180,E1 -19877.946,E2 -19877.946} C_VEL
LIN {X 0,Y 226.648,Z 670.603,A -85,B 0,C 180,E1 -19880.632,E2 -19880.632} C_VEL
LIN {X 0,Y 226.486,Z 676.339,A -85,B 0,C 180,E1 -19883.209,E2 -19883.209} C_VEL
LIN {X 0,Y 226.52,Z 680.432,A -85,B 0,C 180,E1 -19885.552,E2 -19885.552} C_VEL
LIN {X 0,Y 226.609,Z 683.933,A -85,B 0,C 180,E1 -19888.223,E2 -19888.223} C_VEL
LIN {X 0,Y 226.644,Z 685.632,A -85,B 0,C 180,E1 -19890.001,E2 -19890.001} C_VEL
LIN {X 0,Y 226.423,Z 686.795,A -85,B 0,C 180,E1 -19891.779,E2 -19891.779} C_VEL
LIN {X 0,Y 225.972,Z 687.845,A -85,B 0,C 180,E1 -19895.354,E2 -19895.354} C_VEL
LIN {X 0,Y 225.895,Z 687.752,A -85,B 0,C 180,E1 -19897.15,E2 -19897.15} C_VEL
LIN {X 0,Y 226.423,Z 686.324,A -85,B 0,C 180,E1 -19900.734,E2 -19900.734} C_VEL
LIN {X 0,Y 226.927,Z 685.027,A -85,B 0,C 180,E1 -19902.521,E2 -19902.521} C_VEL
LIN {X 0,Y 228.302,Z 682.316,A -85,B 0,C 180,E1 -19905.169,E2 -19905.169} C_VEL
LIN {X 0,Y 230.854,Z 677.253,A -85,B 0,C 180,E1 -19908.643,E2 -19908.643} C_VEL
LIN {X 0,Y 233.46,Z 672.234,A -85,B 0,C 180,E1 -19911.177,E2 -19911.177} C_VEL
LIN {X 0,Y 236.612,Z 666.024,A -85,B 0,C 180,E1 -19913.641,E2 -19913.641} C_VEL
LIN {X 0,Y 240.337,Z 658.513,A -85,B 0,C 180,E1 -19916.018,E2 -19916.018} C_VEL
LIN {X 0,Y 244.63,Z 649.389,A -85,B 0,C 180,E1 -19918.297,E2 -19918.297} C_VEL
LIN {X 0,Y 248.994,Z 639.225,A -85,B 0,C 180,E1 -19920.301,E2 -19920.301} C_VEL
LIN {X 0,Y 253.415,Z 628.029,A -85,B 0,C 180,E1 -19922.033,E2 -19922.033} C_VEL
LIN {X 0,Y 257.32,Z 617.09,A -85,B 0,C 180,E1 -19923.344,E2 -19923.344} C_VEL
LIN {X 0,Y 260.851,Z 605.385,A -85,B 0,C 180,E1 -19924.458,E2 -19924.458} C_VEL
LIN {X 0,Y 264.239,Z 591.411,A -85,B 0,C 180,E1 -19925.462,E2 -19925.462} C_VEL
LIN {X 0,Y 266.872,Z 577.649,A -85,B 0,C 180,E1 -19926.162,E2 -19926.162} C_VEL
LIN {X 0,Y 271.244,Z 543.467,A -85,B 0,C 180,E1 -19927.602,E2 -19927.602} C_VEL
LIN {X 0,Y 271.316,Z 532.128,A -85,B 0,C 180,E1 -19928.599,E2 -19928.599} C_VEL
LIN {X 0,Y 271.194,Z 526.414,A -85,B 0,C 180,E1 -19929.214,E2 -19929.214} C_VEL
LIN {X 0,Y 268.943,Z 519.639,A -85,B 0,C 180,E1 -19930.909,E2 -19930.909} C_VEL
LIN {X 0,Y 267.402,Z 515.398,A -85,B 0,C 180,E1 -19932.239,E2 -19932.239} C_VEL
LIN {X 0,Y 265.682,Z 510.937,A -85,B 0,C 180,E1 -19933.876,E2 -19933.876} C_VEL
LIN {X 0,Y 263.473,Z 505.233,A -85,B 0,C 180,E1 -19936.608,E2 -19936.608} C_VEL
LIN {X 0,Y 261.768,Z 501.278,A -85,B 0,C 180,E1 -19939.882,E2 -19939.882} C_VEL
LIN {X 0,Y 261.314,Z 499.214,A -85,B 0,C 180,E1 -19942.818,E2 -19942.818} C_VEL
LIN {X 0,Y 261.774,Z 498.855,A -85,B 0,C 180,E1 -19945.681,E2 -19945.681} C_VEL
LIN {X 0,Y 263.269,Z 499.581,A -85,B 0,C 180,E1 -19948.477,E2 -19948.477} C_VEL
LIN {X 0,Y 265.81,Z 502.709,A -85,B 0,C 180,E1 -19951.518,E2 -19951.518} C_VEL
LIN {X 0,Y 268.308,Z 506.303,A -85,B 0,C 180,E1 -19953.718,E2 -19953.718} C_VEL
LIN {X 0,Y 270.635,Z 510.075,A -85,B 0,C 180,E1 -19955.449,E2 -19955.449} C_VEL
LIN {X 0,Y 273.145,Z 514.597,A -85,B 0,C 180,E1 -19957.043,E2 -19957.043} C_VEL
LIN {X 0,Y 274.061,Z 516.661,A -85,B 0,C 180,E1 -19957.636,E2 -19957.636} C_VEL
LIN {X 0,Y 268.327,Z 559.76,A -85,B 0,C 180,E1 -19959.443,E2 -19959.443} C_VEL
LIN {X 0,Y 266.299,Z 572.097,A -85,B 0,C 180,E1 -19960.236,E2 -19960.236} C_VEL
LIN {X 0,Y 263.458,Z 584.895,A -85,B 0,C 180,E1 -19961.33,E2 -19961.33} C_VEL
LIN {X 0,Y 260.071,Z 597.223,A -85,B 0,C 180,E1 -19962.707,E2 -19962.707} C_VEL
LIN {X 0,Y 256.672,Z 607.29,A -85,B 0,C 180,E1 -19964.109,E2 -19964.109} C_VEL
LIN {X 0,Y 253.517,Z 615.589,A -85,B 0,C 180,E1 -19965.552,E2 -19965.552} C_VEL
LIN {X 0,Y 249.761,Z 624.349,A -85,B 0,C 180,E1 -19967.404,E2 -19967.404} C_VEL
LIN {X 0,Y 245.561,Z 632.983,A -85,B 0,C 180,E1 -19969.696,E2 -19969.696} C_VEL
LIN {X 0,Y 241.76,Z 639.993,A -85,B 0,C 180,E1 -19972.107,E2 -19972.107} C_VEL
LIN {X 0,Y 237.895,Z 646.278,A -85,B 0,C 180,E1 -19974.915,E2 -19974.915} C_VEL
LIN {X 0,Y 235.037,Z 650.437,A -85,B 0,C 180,E1 -19977.429,E2 -19977.429} C_VEL
LIN {X 0,Y 231.947,Z 654.198,A -85,B 0,C 180,E1 -19980.756,E2 -19980.756} C_VEL
LIN {X 0,Y 229.943,Z 656.05,A -85,B 0,C 180,E1 -19983.504,E2 -19983.504} C_VEL
LIN {X 0,Y 228.887,Z 656.71,A -85,B 0,C 180,E1 -19985.285,E2 -19985.285} C_VEL
LIN {X 0,Y 227.439,Z 656.749,A -85,B 0,C 180,E1 -19988.571,E2 -19988.571} C_VEL
LIN {X 0,Y 226.754,Z 656.034,A -85,B 0,C 180,E1 -19990.717,E2 -19990.717} C_VEL
LIN {X 0,Y 226.358,Z 654.948,A -85,B 0,C 180,E1 -19992.553,E2 -19992.553} C_VEL
LIN {X 0,Y 226.07,Z 652.261,A -85,B 0,C 180,E1 -19995.478,E2 -19995.478} C_VEL
LIN {X 0,Y 226.031,Z 648.816,A -85,B 0,C 180,E1 -19998.115,E2 -19998.115} C_VEL
LIN {X 0,Y 226.392,Z 643.089,A -85,B 0,C 180,E1 -20001.359,E2 -20001.359} C_VEL
LIN {X 0,Y 226.99,Z 636.5,A -85,B 0,C 180,E1 -20004.22,E2 -20004.22} C_VEL
LIN {X 0,Y 227.784,Z 628.887,A -85,B 0,C 180,E1 -20006.843,E2 -20006.843} C_VEL
LIN {X 0,Y 228.838,Z 619.595,A -85,B 0,C 180,E1 -20009.432,E2 -20009.432} C_VEL
LIN {X 0,Y 230.07,Z 608.918,A -85,B 0,C 180,E1 -20011.799,E2 -20011.799} C_VEL
LIN {X 0,Y 231.209,Z 598.373,A -85,B 0,C 180,E1 -20013.693,E2 -20013.693} C_VEL
LIN {X 0,Y 232.499,Z 586.395,A -85,B 0,C 180,E1 -20015.413,E2 -20015.413} C_VEL
LIN {X 0,Y 233.64,Z 573.546,A -85,B 0,C 180,E1 -20016.851,E2 -20016.851} C_VEL
LIN {X 0,Y 234.642,Z 560.362,A -85,B 0,C 180,E1 -20017.948,E2 -20017.948} C_VEL
LIN {X 0,Y 235.223,Z 547.054,A -85,B 0,C 180,E1 -20018.724,E2 -20018.724} C_VEL
LIN {X 0,Y 237.939,Z 484.504,A -85,B 0,C 180,E1 -20021.412,E2 -20021.412} C_VEL
LIN {X 0,Y 227.87,Z 455.099,A -85,B 0,C 180,E1 -20023.503,E2 -20023.503} C_VEL
LIN {X 0,Y 227.803,Z 455.106,A -85,B 0,C 180,E1 -20027.768,E2 -20027.768} C_VEL
LIN {X 0,Y 227.839,Z 455.103,A -85,B 0,C 180,E1 -20031.907,E2 -20031.907} C_VEL
LIN {X 0,Y 227.88,Z 455.099,A -85,B 0,C 180,E1 -20036.377,E2 -20036.377} C_VEL
LIN {X 0,Y 227.878,Z 455.1,A -85,B 0,C 180,E1 -20040.431,E2 -20040.431} C_VEL
LIN {X 0,Y 227.904,Z 455.096,A -85,B 0,C 180,E1 -20044.422,E2 -20044.422} C_VEL
LIN {X 0,Y 227.958,Z 455.091,A -85,B 0,C 180,E1 -20048.286,E2 -20048.286} C_VEL
LIN {X 0,Y 228.037,Z 455.078,A -85,B 0,C 180,E1 -20052.825,E2 -20052.825} C_VEL
LIN {X 0,Y 228.071,Z 455.073,A -85,B 0,C 180,E1 -20057.542,E2 -20057.542} C_VEL
LIN {X 0,Y 228.254,Z 455.049,A -85,B 0,C 180,E1 -20061.143,E2 -20061.143} C_VEL
LIN {X 0,Y 228.303,Z 455.045,A -85,B 0,C 180,E1 -20062.926,E2 -20062.926} C_VEL
LIN {X 0,Y 228.551,Z 455.014,A -85,B 0,C 180,E1 -20068.237,E2 -20068.237} C_VEL
LIN {X 0,Y 228.55,Z 455.013,A -85,B 0,C 180,E1 -20071.762,E2 -20071.762} C_VEL
LIN {X 0,Y 228.319,Z 455.04,A -85,B 0,C 180,E1 -20077.072,E2 -20077.072} C_VEL
LIN {X 0,Y 228.146,Z 455.067,A -85,B 0,C 180,E1 -20080.651,E2 -20080.651} C_VEL
LIN {X 0,Y 228.049,Z 455.078,A -85,B 0,C 180,E1 -20084.272,E2 -20084.272} C_VEL
LIN {X 0,Y 227.969,Z 455.085,A -85,B 0,C 180,E1 -20087.955,E2 -20087.955} C_VEL
LIN {X 0,Y 227.92,Z 455.095,A -85,B 0,C 180,E1 -20092.322,E2 -20092.322} C_VEL
LIN {X 0,Y 227.922,Z 455.094,A -85,B 0,C 180,E1 -20096.592,E2 -20096.592} C_VEL
LIN {X 0,Y 227.873,Z 455.1,A -85,B 0,C 180,E1 -20100.28,E2 -20100.28} C_VEL
LIN {X 0,Y 227.876,Z 455.095,A -85,B 0,C 180,E1 -20103.72,E2 -20103.72} C_VEL
LIN {X 0,Y 227.842,Z 455.103,A -85,B 0,C 180,E1 -20108.091,E2 -20108.091} C_VEL
LIN {X 0,Y 227.798,Z 455.108,A -85,B 0,C 180,E1 -20112.745,E2 -20112.745} C_VEL
LIN {X 0,Y 227.804,Z 455.107,A -85,B 0,C 180,E1 -20117.256,E2 -20117.256} C_VEL
LIN {X 0,Y 227.842,Z 455.099,A -85,B 0,C 180,E1 -20121.909,E2 -20121.909} C_VEL
LIN {X 0,Y 227.878,Z 455.1,A -85,B 0,C 180,E1 -20126.377,E2 -20126.377} C_VEL
LIN {X 0,Y 227.903,Z 455.094,A -85,B 0,C 180,E1 -20130.436,E2 -20130.436} C_VEL
LIN {X 0,Y 227.927,Z 455.094,A -85,B 0,C 180,E1 -20134.426,E2 -20134.426} C_VEL
LIN {X 0,Y 227.961,Z 455.087,A -85,B 0,C 180,E1 -20138.287,E2 -20138.287} C_VEL
LIN {X 0,Y 228.034,Z 455.081,A -85,B 0,C 180,E1 -20142.826,E2 -20142.826} C_VEL
LIN {X 0,Y 228.075,Z 455.069,A -85,B 0,C 180,E1 -20147.543,E2 -20147.543} C_VEL
LIN {X 0,Y 228.304,Z 455.045,A -85,B 0,C 180,E1 -20151.146,E2 -20151.146} C_VEL
LIN {X 0,Y 228.351,Z 455.04,A -85,B 0,C 180,E1 -20152.929,E2 -20152.929} C_VEL
LIN {X 0,Y 228.553,Z 455.013,A -85,B 0,C 180,E1 -20158.238,E2 -20158.238} C_VEL
LIN {X 0,Y 228.554,Z 455.013,A -85,B 0,C 180,E1 -20161.762,E2 -20161.762} C_VEL
LIN {X 0,Y 228.358,Z 455.039,A -85,B 0,C 180,E1 -20167.071,E2 -20167.071} C_VEL
LIN {X 0,Y 228.171,Z 455.064,A -85,B 0,C 180,E1 -20170.65,E2 -20170.65} C_VEL
LIN {X 0,Y 228.057,Z 455.075,A -85,B 0,C 180,E1 -20176.102,E2 -20176.102} C_VEL
LIN {X 0,Y 227.937,Z 455.09,A -85,B 0,C 180,E1 -20179.826,E2 -20179.826} C_VEL
LIN {X 0,Y 227.906,Z 455.092,A -85,B 0,C 180,E1 -20183.634,E2 -20183.634} C_VEL
LIN {X 0,Y 227.886,Z 455.096,A -85,B 0,C 180,E1 -20187.555,E2 -20187.555} C_VEL
LIN {X 0,Y 227.87,Z 455.095,A -85,B 0,C 180,E1 -20191.622,E2 -20191.622} C_VEL
LIN {X 0,Y 227.88,Z 455.097,A -85,B 0,C 180,E1 -20195.872,E2 -20195.872} C_VEL
LIN {X 0,Y 227.826,Z 455.102,A -85,B 0,C 180,E1 -20200.377,E2 -20200.377} C_VEL
LIN {X 0,Y 227.835,Z 455.104,A -85,B 0,C 180,E1 -20205.193,E2 -20205.193} C_VEL
LIN {X 0,Y 227.826,Z 455.102,A -85,B 0,C 180,E1 -20209.624,E2 -20209.624} C_VEL
LIN {X 0,Y 227.984,Z 455.184,A -85,B 0,C 180,E1 -20212.907,E2 -20212.907} C_VEL
LIN {X 0,Y 228.747,Z 458.941,A -85,B 0,C 180,E1 -20214.295,E2 -20214.295} C_VEL
LIN {X 0,Y 228.75,Z 462.38,A -85,B 0,C 180,E1 -20215.496,E2 -20215.496} C_VEL
LIN {X 0,Y 225.289,Z 475.536,A -85,B 0,C 180,E1 -20219.819,E2 -20219.819} C_VEL
LIN {X 0,Y 225.36,Z 477.893,A -85,B 0,C 180,E1 -20220.633,E2 -20220.633} C_VEL
LIN {X 0,Y 225.888,Z 484.229,A -85,B 0,C 180,E1 -20221.009,E2 -20221.009} C_VEL
LIN {X 0,Y 228.405,Z 518.547,A -85,B 0,C 180,E1 -20222.828,E2 -20222.828} C_VEL
LIN {X 0,Y 230.002,Z 536.583,A -85,B 0,C 180,E1 -20223.771,E2 -20223.771} C_VEL
LIN {X 0,Y 227.644,Z 588.253,A -85,B 0,C 180,E1 -20226.157,E2 -20226.157} C_VEL
LIN {X 0,Y 226.733,Z 601.241,A -85,B 0,C 180,E1 -20227.084,E2 -20227.084} C_VEL
LIN {X 0,Y 225.46,Z 613.424,A -85,B 0,C 180,E1 -20228.275,E2 -20228.275} C_VEL
LIN {X 0,Y 224.05,Z 626.571,A -85,B 0,C 180,E1 -20229.99,E2 -20229.99} C_VEL
LIN {X 0,Y 222.757,Z 637.689,A -85,B 0,C 180,E1 -20231.848,E2 -20231.848} C_VEL
LIN {X 0,Y 221.557,Z 647.5,A -85,B 0,C 180,E1 -20233.886,E2 -20233.886} C_VEL
LIN {X 0,Y 220.627,Z 656.514,A -85,B 0,C 180,E1 -20236.178,E2 -20236.178} C_VEL
LIN {X 0,Y 219.96,Z 663.913,A -85,B 0,C 180,E1 -20238.482,E2 -20238.482} C_VEL
LIN {X 0,Y 219.561,Z 671.111,A -85,B 0,C 180,E1 -20241.255,E2 -20241.255} C_VEL
LIN {X 0,Y 219.453,Z 676.328,A -85,B 0,C 180,E1 -20243.781,E2 -20243.781} C_VEL
LIN {X 0,Y 219.535,Z 680.475,A -85,B 0,C 180,E1 -20246.33,E2 -20246.33} C_VEL
LIN {X 0,Y 219.599,Z 682.782,A -85,B 0,C 180,E1 -20248.167,E2 -20248.167} C_VEL
LIN {X 0,Y 219.624,Z 684.597,A -85,B 0,C 180,E1 -20250.001,E2 -20250.001} C_VEL
LIN {X 0,Y 219.36,Z 685.904,A -85,B 0,C 180,E1 -20251.837,E2 -20251.837} C_VEL
LIN {X 0,Y 218.979,Z 686.713,A -85,B 0,C 180,E1 -20253.681,E2 -20253.681} C_VEL
LIN {X 0,Y 218.904,Z 687.13,A -85,B 0,C 180,E1 -20255.574,E2 -20255.574} C_VEL
LIN {X 0,Y 219.013,Z 686.747,A -85,B 0,C 180,E1 -20259.234,E2 -20259.234} C_VEL
LIN {X 0,Y 219.393,Z 685.965,A -85,B 0,C 180,E1 -20261.082,E2 -20261.082} C_VEL
LIN {X 0,Y 220.883,Z 683.188,A -85,B 0,C 180,E1 -20264.747,E2 -20264.747} C_VEL
LIN {X 0,Y 222.693,Z 680.076,A -85,B 0,C 180,E1 -20267.447,E2 -20267.447} C_VEL
LIN {X 0,Y 225.576,Z 674.997,A -85,B 0,C 180,E1 -20270.635,E2 -20270.635} C_VEL
LIN {X 0,Y 228.993,Z 668.914,A -85,B 0,C 180,E1 -20273.515,E2 -20273.515} C_VEL
LIN {X 0,Y 233.351,Z 660.936,A -85,B 0,C 180,E1 -20276.375,E2 -20276.375} C_VEL
LIN {X 0,Y 237.755,Z 652.486,A -85,B 0,C 180,E1 -20278.709,E2 -20278.709} C_VEL
LIN {X 0,Y 242.654,Z 642.321,A -85,B 0,C 180,E1 -20280.938,E2 -20280.938} C_VEL
LIN {X 0,Y 247.117,Z 631.967,A -85,B 0,C 180,E1 -20282.709,E2 -20282.709} C_VEL
LIN {X 0,Y 251.574,Z 620.625,A -85,B 0,C 180,E1 -20284.21,E2 -20284.21} C_VEL
LIN {X 0,Y 255.795,Z 608.277,A -85,B 0,C 180,E1 -20285.48,E2 -20285.48} C_VEL
LIN {X 0,Y 259.566,Z 594.638,A -85,B 0,C 180,E1 -20286.561,E2 -20286.561} C_VEL
LIN {X 0,Y 262.725,Z 579.917,A -85,B 0,C 180,E1 -20287.366,E2 -20287.366} C_VEL
LIN {X 0,Y 267.577,Z 544.931,A -85,B 0,C 180,E1 -20288.867,E2 -20288.867} C_VEL
LIN {X 0,Y 267.87,Z 534.277,A -85,B 0,C 180,E1 -20289.837,E2 -20289.837} C_VEL
LIN {X 0,Y 267.775,Z 530.323,A -85,B 0,C 180,E1 -20290.291,E2 -20290.291} C_VEL
LIN {X 0,Y 265.95,Z 524.357,A -85,B 0,C 180,E1 -20291.894,E2 -20291.894} C_VEL
LIN {X 0,Y 264.368,Z 519.971,A -85,B 0,C 180,E1 -20293.369,E2 -20293.369} C_VEL
LIN {X 0,Y 263.344,Z 516.982,A -85,B 0,C 180,E1 -20294.542,E2 -20294.542} C_VEL
LIN {X 0,Y 261.515,Z 511.64,A -85,B 0,C 180,E1 -20297.131,E2 -20297.131} C_VEL
LIN {X 0,Y 259.946,Z 507.657,A -85,B 0,C 180,E1 -20300.653,E2 -20300.653} C_VEL
LIN {X 0,Y 259.763,Z 506.028,A -85,B 0,C 180,E1 -20303.191,E2 -20303.191} C_VEL
LIN {X 0,Y 260.179,Z 505.781,A -85,B 0,C 180,E1 -20305.441,E2 -20305.441} C_VEL
LIN {X 0,Y 261.547,Z 506.384,A -85,B 0,C 180,E1 -20308.246,E2 -20308.246} C_VEL
LIN {X 0,Y 263.832,Z 509.312,A -85,B 0,C 180,E1 -20311.16,E2 -20311.16} C_VEL
LIN {X 0,Y 266.109,Z 512.809,A -85,B 0,C 180,E1 -20313.322,E2 -20313.322} C_VEL
LIN {X 0,Y 269.066,Z 517.808,A -85,B 0,C 180,E1 -20315.569,E2 -20315.569} C_VEL
LIN {X 0,Y 270.349,Z 520.626,A -85,B 0,C 180,E1 -20316.453,E2 -20316.453} C_VEL
LIN {X 0,Y 264.665,Z 560.26,A -85,B 0,C 180,E1 -20318.136,E2 -20318.136} C_VEL
LIN {X 0,Y 262.331,Z 573.607,A -85,B 0,C 180,E1 -20319.003,E2 -20319.003} C_VEL
LIN {X 0,Y 259.571,Z 585.406,A -85,B 0,C 180,E1 -20320.012,E2 -20320.012} C_VEL
LIN {X 0,Y 255.977,Z 597.651,A -85,B 0,C 180,E1 -20321.387,E2 -20321.387} C_VEL
LIN {X 0,Y 251.943,Z 608.78,A -85,B 0,C 180,E1 -20322.968,E2 -20322.968} C_VEL
LIN {X 0,Y 248.211,Z 617.983,A -85,B 0,C 180,E1 -20324.615,E2 -20324.615} C_VEL
LIN {X 0,Y 243.877,Z 627.14,A -85,B 0,C 180,E1 -20326.671,E2 -20326.671} C_VEL
LIN {X 0,Y 239.47,Z 635.307,A -85,B 0,C 180,E1 -20329.003,E2 -20329.003} C_VEL
LIN {X 0,Y 235.561,Z 641.93,A -85,B 0,C 180,E1 -20331.421,E2 -20331.421} C_VEL
LIN {X 0,Y 231.986,Z 647.191,A -85,B 0,C 180,E1 -20333.913,E2 -20333.913} C_VEL
LIN {X 0,Y 228.868,Z 651.261,A -85,B 0,C 180,E1 -20336.479,E2 -20336.479} C_VEL
LIN {X 0,Y 227.07,Z 653.388,A -85,B 0,C 180,E1 -20338.226,E2 -20338.226} C_VEL
LIN {X 0,Y 224.912,Z 655.558,A -85,B 0,C 180,E1 -20340.619,E2 -20340.619} C_VEL
LIN {X 0,Y 222.761,Z 657.124,A -85,B 0,C 180,E1 -20343.618,E2 -20343.618} C_VEL
LIN {X 0,Y 221.676,Z 657.518,A -85,B 0,C 180,E1 -20345.458,E2 -20345.458} C_VEL
LIN {X 0,Y 220.339,Z 657.232,A -85,B 0,C 180,E1 -20348.583,E2 -20348.583} C_VEL
LIN {X 0,Y 219.567,Z 656.134,A -85,B 0,C 180,E1 -20351.072,E2 -20351.072} C_VEL
LIN {X 0,Y 219.203,Z 654.808,A -85,B 0,C 180,E1 -20352.969,E2 -20352.969} C_VEL
LIN {X 0,Y 218.963,Z 652.139,A -85,B 0,C 180,E1 -20355.653,E2 -20355.653} C_VEL
LIN {X 0,Y 218.969,Z 647.927,A -85,B 0,C 180,E1 -20358.721,E2 -20358.721} C_VEL
LIN {X 0,Y 219.34,Z 642.462,A -85,B 0,C 180,E1 -20361.687,E2 -20361.687} C_VEL
LIN {X 0,Y 219.963,Z 635.756,A -85,B 0,C 180,E1 -20364.542,E2 -20364.542} C_VEL
LIN {X 0,Y 220.751,Z 628.237,A -85,B 0,C 180,E1 -20367.128,E2 -20367.128} C_VEL
LIN {X 0,Y 221.711,Z 620.097,A -85,B 0,C 180,E1 -20369.428,E2 -20369.428} C_VEL
LIN {X 0,Y 222.928,Z 609.557,A -85,B 0,C 180,E1 -20371.849,E2 -20371.849} C_VEL
LIN {X 0,Y 224.117,Z 598.963,A -85,B 0,C 180,E1 -20373.822,E2 -20373.822} C_VEL
LIN {X 0,Y 225.365,Z 587.752,A -85,B 0,C 180,E1 -20375.508,E2 -20375.508} C_VEL
LIN {X 0,Y 226.586,Z 574.343,A -85,B 0,C 180,E1 -20377.077,E2 -20377.077} C_VEL
LIN {X 0,Y 227.586,Z 561.25,A -85,B 0,C 180,E1 -20378.212,E2 -20378.212} C_VEL
LIN {X 0,Y 228.275,Z 547.045,A -85,B 0,C 180,E1 -20379.063,E2 -20379.063} C_VEL
LIN {X 0,Y 231.026,Z 485.922,A -85,B 0,C 180,E1 -20381.778,E2 -20381.778} C_VEL
LIN {X 0,Y 220.806,Z 455.98,A -85,B 0,C 180,E1 -20383.951,E2 -20383.951} C_VEL
LIN {X 0,Y 220.761,Z 455.984,A -85,B 0,C 180,E1 -20388.044,E2 -20388.044} C_VEL
LIN {X 0,Y 220.827,Z 455.975,A -85,B 0,C 180,E1 -20392.792,E2 -20392.792} C_VEL
LIN {X 0,Y 220.814,Z 455.977,A -85,B 0,C 180,E1 -20397.243,E2 -20397.243} C_VEL
LIN {X 0,Y 220.806,Z 455.977,A -85,B 0,C 180,E1 -20401.481,E2 -20401.481} C_VEL
LIN {X 0,Y 220.85,Z 455.972,A -85,B 0,C 180,E1 -20405.562,E2 -20405.562} C_VEL
LIN {X 0,Y 220.89,Z 455.967,A -85,B 0,C 180,E1 -20409.513,E2 -20409.513} C_VEL
LIN {X 0,Y 221.019,Z 455.951,A -85,B 0,C 180,E1 -20413.37,E2 -20413.37} C_VEL
LIN {X 0,Y 221.068,Z 455.944,A -85,B 0,C 180,E1 -20419.003,E2 -20419.003} C_VEL
LIN {X 0,Y 221.241,Z 455.926,A -85,B 0,C 180,E1 -20422.699,E2 -20422.699} C_VEL
LIN {X 0,Y 221.509,Z 455.891,A -85,B 0,C 180,E1 -20428.181,E2 -20428.181} C_VEL
LIN {X 0,Y 221.507,Z 455.891,A -85,B 0,C 180,E1 -20431.818,E2 -20431.818} C_VEL
LIN {X 0,Y 221.255,Z 455.919,A -85,B 0,C 180,E1 -20437.299,E2 -20437.299} C_VEL
LIN {X 0,Y 221.067,Z 455.947,A -85,B 0,C 180,E1 -20440.996,E2 -20440.996} C_VEL
LIN {X 0,Y 220.977,Z 455.957,A -85,B 0,C 180,E1 -20444.739,E2 -20444.739} C_VEL
LIN {X 0,Y 220.899,Z 455.969,A -85,B 0,C 180,E1 -20448.551,E2 -20448.551} C_VEL
LIN {X 0,Y 220.867,Z 455.972,A -85,B 0,C 180,E1 -20452.664,E2 -20452.664} C_VEL
LIN {X 0,Y 220.865,Z 455.971,A -85,B 0,C 180,E1 -20457.005,E2 -20457.005} C_VEL
LIN {X 0,Y 220.817,Z 455.979,A -85,B 0,C 180,E1 -20460.758,E2 -20460.758} C_VEL
LIN {X 0,Y 220.8,Z 455.979,A -85,B 0,C 180,E1 -20464.954,E2 -20464.954} C_VEL
LIN {X 0,Y 220.809,Z 455.978,A -85,B 0,C 180,E1 -20467.277,E2 -20467.277} C_VEL
LIN {X 0,Y 220.757,Z 455.983,A -85,B 0,C 180,E1 -20471.955,E2 -20471.955} C_VEL
LIN {X 0,Y 220.765,Z 455.983,A -85,B 0,C 180,E1 -20475.544,E2 -20475.544} C_VEL
LIN {X 0,Y 220.805,Z 455.98,A -85,B 0,C 180,E1 -20480.463,E2 -20480.463} C_VEL
LIN {X 0,Y 220.8,Z 455.98,A -85,B 0,C 180,E1 -20485.045,E2 -20485.045} C_VEL
LIN {X 0,Y 220.833,Z 455.972,A -85,B 0,C 180,E1 -20489.389,E2 -20489.389} C_VEL
LIN {X 0,Y 220.893,Z 455.967,A -85,B 0,C 180,E1 -20493.549,E2 -20493.549} C_VEL
LIN {X 0,Y 220.877,Z 455.968,A -85,B 0,C 180,E1 -20497.553,E2 -20497.553} C_VEL
LIN {X 0,Y 220.984,Z 455.96,A -85,B 0,C 180,E1 -20502.571,E2 -20502.571} C_VEL
LIN {X 0,Y 221.013,Z 455.95,A -85,B 0,C 180,E1 -20507.139,E2 -20507.139} C_VEL
LIN {X 0,Y 221.235,Z 455.927,A -85,B 0,C 180,E1 -20510.861,E2 -20510.861} C_VEL
LIN {X 0,Y 221.302,Z 455.92,A -85,B 0,C 180,E1 -20512.702,E2 -20512.702} C_VEL
LIN {X 0,Y 221.511,Z 455.89,A -85,B 0,C 180,E1 -20518.182,E2 -20518.182} C_VEL
LIN {X 0,Y 221.512,Z 455.89,A -85,B 0,C 180,E1 -20521.818,E2 -20521.818} C_VEL
LIN {X 0,Y 221.295,Z 455.917,A -85,B 0,C 180,E1 -20527.298,E2 -20527.298} C_VEL
LIN {X 0,Y 221.116,Z 455.941,A -85,B 0,C 180,E1 -20530.994,E2 -20530.994} C_VEL
LIN {X 0,Y 221.016,Z 455.955,A -85,B 0,C 180,E1 -20536.63,E2 -20536.63} C_VEL
LIN {X 0,Y 220.884,Z 455.971,A -85,B 0,C 180,E1 -20540.487,E2 -20540.487} C_VEL
LIN {X 0,Y 220.862,Z 455.972,A -85,B 0,C 180,E1 -20544.436,E2 -20544.436} C_VEL
LIN {X 0,Y 220.836,Z 455.977,A -85,B 0,C 180,E1 -20548.514,E2 -20548.514} C_VEL
LIN {X 0,Y 220.817,Z 455.978,A -85,B 0,C 180,E1 -20552.756,E2 -20552.756} C_VEL
LIN {X 0,Y 220.81,Z 455.978,A -85,B 0,C 180,E1 -20557.279,E2 -20557.279} C_VEL
LIN {X 0,Y 220.77,Z 455.982,A -85,B 0,C 180,E1 -20561.953,E2 -20561.953} C_VEL
LIN {X 0,Y 220.775,Z 455.982,A -85,B 0,C 180,E1 -20565.547,E2 -20565.547} C_VEL
LIN {X 0,Y 220.808,Z 455.978,A -85,B 0,C 180,E1 -20570.464,E2 -20570.464} C_VEL
LIN {X 0,Y 220.928,Z 456.079,A -85,B 0,C 180,E1 -20572.627,E2 -20572.627} C_VEL
LIN {X 0,Y 223.338,Z 468.106,A -85,B 0,C 180,E1 -20577.125,E2 -20577.125} C_VEL
LIN {X 0,Y 225.36,Z 477.893,A -85,B 0,C 180,E1 -20580.633,E2 -20580.633} C_VEL
LIN {X 0,Y 223.579,Z 482.434,A -85,B 0,C 180,E1 -20580.765,E2 -20580.765} C_VEL
LIN {X 0,Y 219.411,Z 492.273,A -85,B 0,C 180,E1 -20580.951,E2 -20580.951} C_VEL
LIN {X 0,Y 219.057,Z 495.99,A -85,B 0,C 180,E1 -20581.041,E2 -20581.041} C_VEL
LIN {X 0,Y 219.384,Z 500.204,A -85,B 0,C 180,E1 -20581.285,E2 -20581.285} C_VEL
LIN {X 0,Y 220.612,Z 508.684,A -85,B 0,C 180,E1 -20581.872,E2 -20581.872} C_VEL
LIN {X 0,Y 223.039,Z 537.789,A -85,B 0,C 180,E1 -20583.456,E2 -20583.456} C_VEL
LIN {X 0,Y 220.669,Z 587.851,A -85,B 0,C 180,E1 -20585.855,E2 -20585.855} C_VEL
LIN {X 0,Y 219.742,Z 600.775,A -85,B 0,C 180,E1 -20586.81,E2 -20586.81} C_VEL
LIN {X 0,Y 218.452,Z 612.873,A -85,B 0,C 180,E1 -20588.038,E2 -20588.038} C_VEL
LIN {X 0,Y 216.988,Z 626.268,A -85,B 0,C 180,E1 -20589.856,E2 -20589.856} C_VEL
LIN {X 0,Y 215.72,Z 637.041,A -85,B 0,C 180,E1 -20591.726,E2 -20591.726} C_VEL
LIN {X 0,Y 214.511,Z 646.824,A -85,B 0,C 180,E1 -20593.831,E2 -20593.831} C_VEL
LIN {X 0,Y 213.573,Z 655.816,A -85,B 0,C 180,E1 -20596.198,E2 -20596.198} C_VEL
LIN {X 0,Y 212.913,Z 663.227,A -85,B 0,C 180,E1 -20598.578,E2 -20598.578} C_VEL
LIN {X 0,Y 212.534,Z 670.454,A -85,B 0,C 180,E1 -20601.443,E2 -20601.443} C_VEL
LIN {X 0,Y 212.437,Z 676.114,A -85,B 0,C 180,E1 -20604.305,E2 -20604.305} C_VEL
LIN {X 0,Y 212.552,Z 680.443,A -85,B 0,C 180,E1 -20607.158,E2 -20607.158} C_VEL
LIN {X 0,Y 212.601,Z 683.537,A -85,B 0,C 180,E1 -20610.001,E2 -20610.001} C_VEL
LIN {X 0,Y 212.315,Z 684.921,A -85,B 0,C 180,E1 -20611.898,E2 -20611.898} C_VEL
LIN {X 0,Y 211.857,Z 686.38,A -85,B 0,C 180,E1 -20615.613,E2 -20615.613} C_VEL
LIN {X 0,Y 211.795,Z 686.493,A -85,B 0,C 180,E1 -20617.628,E2 -20617.628} C_VEL
LIN {X 0,Y 212.381,Z 685.54,A -85,B 0,C 180,E1 -20621.453,E2 -20621.453} C_VEL
LIN {X 0,Y 213.002,Z 684.499,A -85,B 0,C 180,E1 -20623.355,E2 -20623.355} C_VEL
LIN {X 0,Y 213.988,Z 683.063,A -85,B 0,C 180,E1 -20625.234,E2 -20625.234} C_VEL
LIN {X 0,Y 216.614,Z 678.94,A -85,B 0,C 180,E1 -20628.933,E2 -20628.933} C_VEL
LIN {X 0,Y 219.399,Z 674.607,A -85,B 0,C 180,E1 -20631.726,E2 -20631.726} C_VEL
LIN {X 0,Y 222.552,Z 669.56,A -85,B 0,C 180,E1 -20634.239,E2 -20634.239} C_VEL
LIN {X 0,Y 227.088,Z 661.997,A -85,B 0,C 180,E1 -20637.161,E2 -20637.161} C_VEL
LIN {X 0,Y 231.667,Z 654.036,A -85,B 0,C 180,E1 -20639.537,E2 -20639.537} C_VEL
LIN {X 0,Y 236.73,Z 644.302,A -85,B 0,C 180,E1 -20641.801,E2 -20641.801} C_VEL
LIN {X 0,Y 241.837,Z 633.577,A -85,B 0,C 180,E1 -20643.766,E2 -20643.766} C_VEL
LIN {X 0,Y 246.436,Z 622.847,A -85,B 0,C 180,E1 -20645.276,E2 -20645.276} C_VEL
LIN {X 0,Y 251.373,Z 609.562,A -85,B 0,C 180,E1 -20646.7,E2 -20646.7} C_VEL
LIN {X 0,Y 255.863,Z 594.384,A -85,B 0,C 180,E1 -20647.923,E2 -20647.923} C_VEL
LIN {X 0,Y 259.099,Z 580.552,A -85,B 0,C 180,E1 -20648.693,E2 -20648.693} C_VEL
LIN {X 0,Y 263.341,Z 552.602,A -85,B 0,C 180,E1 -20649.896,E2 -20649.896} C_VEL
LIN {X 0,Y 264.253,Z 545.678,A -85,B 0,C 180,E1 -20650.229,E2 -20650.229} C_VEL
LIN {X 0,Y 264.594,Z 535.95,A -85,B 0,C 180,E1 -20651.179,E2 -20651.179} C_VEL
LIN {X 0,Y 264.563,Z 534.532,A -85,B 0,C 180,E1 -20651.37,E2 -20651.37} C_VEL
LIN {X 0,Y 262.739,Z 528.138,A -85,B 0,C 180,E1 -20653.205,E2 -20653.205} C_VEL
LIN {X 0,Y 261.144,Z 523.206,A -85,B 0,C 180,E1 -20655.108,E2 -20655.108} C_VEL
LIN {X 0,Y 259.651,Z 518.299,A -85,B 0,C 180,E1 -20657.505,E2 -20657.505} C_VEL
LIN {X 0,Y 258.336,Z 514.294,A -85,B 0,C 180,E1 -20661.078,E2 -20661.078} C_VEL
LIN {X 0,Y 258.221,Z 512.967,A -85,B 0,C 180,E1 -20663.218,E2 -20663.218} C_VEL
LIN {X 0,Y 258.943,Z 512.812,A -85,B 0,C 180,E1 -20666.26,E2 -20666.26} C_VEL
LIN {X 0,Y 259.93,Z 513.334,A -85,B 0,C 180,E1 -20668.18,E2 -20668.18} C_VEL
LIN {X 0,Y 262.007,Z 516.191,A -85,B 0,C 180,E1 -20670.964,E2 -20670.964} C_VEL
LIN {X 0,Y 264.086,Z 519.518,A -85,B 0,C 180,E1 -20673.032,E2 -20673.032} C_VEL
LIN {X 0,Y 266.778,Z 524.461,A -85,B 0,C 180,E1 -20675.203,E2 -20675.203} C_VEL
LIN {X 0,Y 261.037,Z 562.777,A -85,B 0,C 180,E1 -20676.878,E2 -20676.878} C_VEL
LIN {X 0,Y 258.516,Z 575.693,A -85,B 0,C 180,E1 -20677.753,E2 -20677.753} C_VEL
LIN {X 0,Y 255.455,Z 587.562,A -85,B 0,C 180,E1 -20678.812,E2 -20678.812} C_VEL
LIN {X 0,Y 251.138,Z 600.939,A -85,B 0,C 180,E1 -20680.378,E2 -20680.378} C_VEL
LIN {X 0,Y 246.93,Z 611.594,A -85,B 0,C 180,E1 -20681.97,E2 -20681.97} C_VEL
LIN {X 0,Y 242.801,Z 620.71,A -85,B 0,C 180,E1 -20683.711,E2 -20683.711} C_VEL
LIN {X 0,Y 238.123,Z 629.779,A -85,B 0,C 180,E1 -20685.864,E2 -20685.864} C_VEL
LIN {X 0,Y 233.405,Z 637.706,A -85,B 0,C 180,E1 -20688.273,E2 -20688.273} C_VEL
LIN {X 0,Y 228.658,Z 644.819,A -85,B 0,C 180,E1 -20691.16,E2 -20691.16} C_VEL
LIN {X 0,Y 224.988,Z 649.632,A -85,B 0,C 180,E1 -20693.723,E2 -20693.723} C_VEL
LIN {X 0,Y 221.803,Z 653.281,A -85,B 0,C 180,E1 -20696.367,E2 -20696.367} C_VEL
LIN {X 0,Y 219.937,Z 655.109,A -85,B 0,C 180,E1 -20698.169,E2 -20698.169} C_VEL
LIN {X 0,Y 217.878,Z 656.823,A -85,B 0,C 180,E1 -20700.473,E2 -20700.473} C_VEL
LIN {X 0,Y 215.55,Z 658.096,A -85,B 0,C 180,E1 -20703.739,E2 -20703.739} C_VEL
LIN {X 0,Y 214.456,Z 658.227,A -85,B 0,C 180,E1 -20705.642,E2 -20705.642} C_VEL
LIN {X 0,Y 213.237,Z 657.629,A -85,B 0,C 180,E1 -20708.594,E2 -20708.594} C_VEL
LIN {X 0,Y 212.37,Z 656.119,A -85,B 0,C 180,E1 -20711.453,E2 -20711.453} C_VEL
LIN {X 0,Y 211.948,Z 653.558,A -85,B 0,C 180,E1 -20714.4,E2 -20714.4} C_VEL
LIN {X 0,Y 211.809,Z 649.896,A -85,B 0,C 180,E1 -20717.375,E2 -20717.375} C_VEL
LIN {X 0,Y 212.066,Z 645.021,A -85,B 0,C 180,E1 -20720.364,E2 -20720.364} C_VEL
LIN {X 0,Y 212.583,Z 638.745,A -85,B 0,C 180,E1 -20723.373,E2 -20723.373} C_VEL
LIN {X 0,Y 213.235,Z 632.205,A -85,B 0,C 180,E1 -20725.894,E2 -20725.894} C_VEL
LIN {X 0,Y 214.128,Z 624.246,A -85,B 0,C 180,E1 -20728.419,E2 -20728.419} C_VEL
LIN {X 0,Y 215.27,Z 614.437,A -85,B 0,C 180,E1 -20730.944,E2 -20730.944} C_VEL
LIN {X 0,Y 216.526,Z 604.162,A -85,B 0,C 180,E1 -20733.098,E2 -20733.098} C_VEL
LIN {X 0,Y 217.74,Z 593.281,A -85,B 0,C 180,E1 -20734.954,E2 -20734.954} C_VEL
LIN {X 0,Y 219.023,Z 580.617,A -85,B 0,C 180,E1 -20736.658,E2 -20736.658} C_VEL
LIN {X 0,Y 220.065,Z 568.376,A -85,B 0,C 180,E1 -20737.935,E2 -20737.935} C_VEL
LIN {X 0,Y 221.015,Z 553.93,A -85,B 0,C 180,E1 -20739.014,E2 -20739.014} C_VEL
LIN {X 0,Y 224.165,Z 487.375,A -85,B 0,C 180,E1 -20742.161,E2 -20742.161} C_VEL
LIN {X 0,Y 213.759,Z 456.86,A -85,B 0,C 180,E1 -20744.432,E2 -20744.432} C_VEL
LIN {X 0,Y 213.709,Z 456.863,A -85,B 0,C 180,E1 -20749.146,E2 -20749.146} C_VEL
LIN {X 0,Y 213.743,Z 456.856,A -85,B 0,C 180,E1 -20753.71,E2 -20753.71} C_VEL
LIN {X 0,Y 213.76,Z 456.859,A -85,B 0,C 180,E1 -20758.26,E2 -20758.26} C_VEL
LIN {X 0,Y 213.79,Z 456.852,A -85,B 0,C 180,E1 -20762.597,E2 -20762.597} C_VEL
LIN {X 0,Y 213.813,Z 456.85,A -85,B 0,C 180,E1 -20766.978,E2 -20766.978} C_VEL
LIN {X 0,Y 213.946,Z 456.833,A -85,B 0,C 180,E1 -20772.803,E2 -20772.803} C_VEL
LIN {X 0,Y 213.953,Z 456.834,A -85,B 0,C 180,E1 -20776.706,E2 -20776.706} C_VEL
LIN {X 0,Y 214.135,Z 456.809,A -85,B 0,C 180,E1 -20780.554,E2 -20780.554} C_VEL
LIN {X 0,Y 214.085,Z 456.818,A -85,B 0,C 180,E1 -20784.347,E2 -20784.347} C_VEL
LIN {X 0,Y 214.442,Z 456.771,A -85,B 0,C 180,E1 -20788.121,E2 -20788.121} C_VEL
LIN {X 0,Y 214.54,Z 456.757,A -85,B 0,C 180,E1 -20789.999,E2 -20789.999} C_VEL
LIN {X 0,Y 214.44,Z 456.771,A -85,B 0,C 180,E1 -20791.877,E2 -20791.877} C_VEL
LIN {X 0,Y 214.194,Z 456.798,A -85,B 0,C 180,E1 -20797.541,E2 -20797.541} C_VEL
LIN {X 0,Y 213.998,Z 456.827,A -85,B 0,C 180,E1 -20801.364,E2 -20801.364} C_VEL
LIN {X 0,Y 213.913,Z 456.835,A -85,B 0,C 180,E1 -20805.238,E2 -20805.238} C_VEL
LIN {X 0,Y 213.82,Z 456.849,A -85,B 0,C 180,E1 -20809.188,E2 -20809.188} C_VEL
LIN {X 0,Y 213.802,Z 456.85,A -85,B 0,C 180,E1 -20813.231,E2 -20813.231} C_VEL
LIN {X 0,Y 213.787,Z 456.852,A -85,B 0,C 180,E1 -20817.427,E2 -20817.427} C_VEL
LIN {X 0,Y 213.758,Z 456.856,A -85,B 0,C 180,E1 -20821.738,E2 -20821.738} C_VEL
LIN {X 0,Y 213.743,Z 456.859,A -85,B 0,C 180,E1 -20826.288,E2 -20826.288} C_VEL
LIN {X 0,Y 213.701,Z 456.862,A -85,B 0,C 180,E1 -20831.127,E2 -20831.127} C_VEL
LIN {X 0,Y 213.701,Z 456.861,A -85,B 0,C 180,E1 -20833.679,E2 -20833.679} C_VEL
LIN {X 0,Y 213.701,Z 456.865,A -85,B 0,C 180,E1 -20836.345,E2 -20836.345} C_VEL
LIN {X 0,Y 213.715,Z 456.861,A -85,B 0,C 180,E1 -20839.143,E2 -20839.143} C_VEL
LIN {X 0,Y 213.742,Z 456.857,A -85,B 0,C 180,E1 -20843.711,E2 -20843.711} C_VEL
LIN {X 0,Y 213.779,Z 456.854,A -85,B 0,C 180,E1 -20848.731,E2 -20848.731} C_VEL
LIN {X 0,Y 213.825,Z 456.85,A -85,B 0,C 180,E1 -20852.603,E2 -20852.603} C_VEL
LIN {X 0,Y 213.851,Z 456.844,A -85,B 0,C 180,E1 -20856.953,E2 -20856.953} C_VEL
LIN {X 0,Y 213.932,Z 456.836,A -85,B 0,C 180,E1 -20862.305,E2 -20862.305} C_VEL
LIN {X 0,Y 213.954,Z 456.831,A -85,B 0,C 180,E1 -20866.707,E2 -20866.707} C_VEL
LIN {X 0,Y 214.166,Z 456.808,A -85,B 0,C 180,E1 -20870.556,E2 -20870.556} C_VEL
LIN {X 0,Y 214.238,Z 456.799,A -85,B 0,C 180,E1 -20872.46,E2 -20872.46} C_VEL
LIN {X 0,Y 214.444,Z 456.77,A -85,B 0,C 180,E1 -20878.122,E2 -20878.122} C_VEL
LIN {X 0,Y 214.55,Z 456.758,A -85,B 0,C 180,E1 -20880,E2 -20880} C_VEL
LIN {X 0,Y 214.445,Z 456.771,A -85,B 0,C 180,E1 -20881.878,E2 -20881.878} C_VEL
LIN {X 0,Y 214.235,Z 456.796,A -85,B 0,C 180,E1 -20887.54,E2 -20887.54} C_VEL
LIN {X 0,Y 214.047,Z 456.82,A -85,B 0,C 180,E1 -20891.362,E2 -20891.362} C_VEL
LIN {X 0,Y 213.933,Z 456.834,A -85,B 0,C 180,E1 -20895.237,E2 -20895.237} C_VEL
LIN {X 0,Y 213.835,Z 456.847,A -85,B 0,C 180,E1 -20899.188,E2 -20899.188} C_VEL
LIN {X 0,Y 213.81,Z 456.849,A -85,B 0,C 180,E1 -20903.231,E2 -20903.231} C_VEL
LIN {X 0,Y 213.828,Z 456.848,A -85,B 0,C 180,E1 -20907.45,E2 -20907.45} C_VEL
LIN {X 0,Y 213.776,Z 456.851,A -85,B 0,C 180,E1 -20911.736,E2 -20911.736} C_VEL
LIN {X 0,Y 213.743,Z 456.86,A -85,B 0,C 180,E1 -20916.289,E2 -20916.289} C_VEL
LIN {X 0,Y 213.712,Z 456.862,A -85,B 0,C 180,E1 -20921.126,E2 -20921.126} C_VEL
LIN {X 0,Y 213.707,Z 456.863,A -85,B 0,C 180,E1 -20923.679,E2 -20923.679} C_VEL
LIN {X 0,Y 213.707,Z 456.864,A -85,B 0,C 180,E1 -20926.344,E2 -20926.344} C_VEL
LIN {X 0,Y 213.799,Z 456.851,A -85,B 0,C 180,E1 -20931.35,E2 -20931.35} C_VEL
LIN {X 0,Y 213.877,Z 456.912,A -85,B 0,C 180,E1 -20932.321,E2 -20932.321} C_VEL
LIN {X 0,Y 215.956,Z 467.492,A -85,B 0,C 180,E1 -20936.411,E2 -20936.411} C_VEL
LIN {X 0,Y 218.053,Z 477.607,A -85,B 0,C 180,E1 -20940.132,E2 -20940.132} C_VEL
LIN {X 0,Y 218.907,Z 481.621,A -85,B 0,C 180,E1 -20940.397,E2 -20940.397} C_VEL
LIN {X 0,Y 220.612,Z 508.684,A -85,B 0,C 180,E1 -20941.872,E2 -20941.872} C_VEL
LIN {X 0,Y 220.49,Z 514.48,A -85,B 0,C 180,E1 -20942.152,E2 -20942.152} C_VEL
LIN {X 0,Y 216.349,Z 535.659,A -85,B 0,C 180,E1 -20942.983,E2 -20942.983} C_VEL
LIN {X 0,Y 216.01,Z 539.554,A -85,B 0,C 180,E1 -20943.165,E2 -20943.165} C_VEL
LIN {X 0,Y 213.646,Z 587.696,A -85,B 0,C 180,E1 -20945.592,E2 -20945.592} C_VEL
LIN {X 0,Y 212.643,Z 601.057,A -85,B 0,C 180,E1 -20946.634,E2 -20946.634} C_VEL
LIN {X 0,Y 211.269,Z 613.836,A -85,B 0,C 180,E1 -20948.023,E2 -20948.023} C_VEL
LIN {X 0,Y 209.8,Z 626.818,A -85,B 0,C 180,E1 -20949.886,E2 -20949.886} C_VEL
LIN {X 0,Y 208.406,Z 638.602,A -85,B 0,C 180,E1 -20952.079,E2 -20952.079} C_VEL
LIN {X 0,Y 207.22,Z 648.041,A -85,B 0,C 180,E1 -20954.258,E2 -20954.258} C_VEL
LIN {X 0,Y 206.36,Z 656.726,A -85,B 0,C 180,E1 -20956.71,E2 -20956.71} C_VEL
LIN {X 0,Y 205.717,Z 665.137,A -85,B 0,C 180,E1 -20959.668,E2 -20959.668} C_VEL
LIN {X 0,Y 205.447,Z 672.135,A -85,B 0,C 180,E1 -20962.77,E2 -20962.77} C_VEL
LIN {X 0,Y 205.438,Z 676.256,A -85,B 0,C 180,E1 -20965.095,E2 -20965.095} C_VEL
LIN {X 0,Y 205.578,Z 680.354,A -85,B 0,C 180,E1 -20968.042,E2 -20968.042} C_VEL
LIN {X 0,Y 205.579,Z 682.416,A -85,B 0,C 180,E1 -20970.001,E2 -20970.001} C_VEL
LIN {X 0,Y 205.29,Z 683.905,A -85,B 0,C 180,E1 -20971.963,E2 -20971.963} C_VEL
LIN {X 0,Y 204.802,Z 685.59,A -85,B 0,C 180,E1 -20975.91,E2 -20975.91} C_VEL
LIN {X 0,Y 204.761,Z 685.83,A -85,B 0,C 180,E1 -20977.892,E2 -20977.892} C_VEL
LIN {X 0,Y 204.968,Z 685.668,A -85,B 0,C 180,E1 -20979.872,E2 -20979.872} C_VEL
LIN {X 0,Y 206.062,Z 684.17,A -85,B 0,C 180,E1 -20983.813,E2 -20983.813} C_VEL
LIN {X 0,Y 208.4,Z 681.185,A -85,B 0,C 180,E1 -20987.669,E2 -20987.669} C_VEL
LIN {X 0,Y 210.797,Z 677.88,A -85,B 0,C 180,E1 -20990.493,E2 -20990.493} C_VEL
LIN {X 0,Y 213.777,Z 673.606,A -85,B 0,C 180,E1 -20993.236,E2 -20993.236} C_VEL
LIN {X 0,Y 217.442,Z 668.33,A -85,B 0,C 180,E1 -20995.871,E2 -20995.871} C_VEL
LIN {X 0,Y 221.645,Z 661.885,A -85,B 0,C 180,E1 -20998.401,E2 -20998.401} C_VEL
LIN {X 0,Y 226.468,Z 654.052,A -85,B 0,C 180,E1 -21000.801,E2 -21000.801} C_VEL
LIN {X 0,Y 231.812,Z 644.648,A -85,B 0,C 180,E1 -21003.075,E2 -21003.075} C_VEL
LIN {X 0,Y 237.168,Z 634.131,A -85,B 0,C 180,E1 -21005.04,E2 -21005.04} C_VEL
LIN {X 0,Y 242.53,Z 622.444,A -85,B 0,C 180,E1 -21006.704,E2 -21006.704} C_VEL
LIN {X 0,Y 247.661,Z 609.45,A -85,B 0,C 180,E1 -21008.114,E2 -21008.114} C_VEL
LIN {X 0,Y 252.04,Z 595.685,A -85,B 0,C 180,E1 -21009.245,E2 -21009.245} C_VEL
LIN {X 0,Y 255.627,Z 581.569,A -85,B 0,C 180,E1 -21010.055,E2 -21010.055} C_VEL
LIN {X 0,Y 259.566,Z 558.046,A -85,B 0,C 180,E1 -21011.083,E2 -21011.083} C_VEL
LIN {X 0,Y 261.086,Z 548.035,A -85,B 0,C 180,E1 -21011.521,E2 -21011.521} C_VEL
LIN {X 0,Y 261.579,Z 539.027,A -85,B 0,C 180,E1 -21012.412,E2 -21012.412} C_VEL
LIN {X 0,Y 260.157,Z 533.43,A -85,B 0,C 180,E1 -21014.129,E2 -21014.129} C_VEL
LIN {X 0,Y 258.926,Z 529.268,A -85,B 0,C 180,E1 -21015.772,E2 -21015.772} C_VEL
LIN {X 0,Y 257.728,Z 524.766,A -85,B 0,C 180,E1 -21018.01,E2 -21018.01} C_VEL
LIN {X 0,Y 256.731,Z 521.07,A -85,B 0,C 180,E1 -21021.422,E2 -21021.422} C_VEL
LIN {X 0,Y 256.765,Z 519.748,A -85,B 0,C 180,E1 -21023.822,E2 -21023.822} C_VEL
LIN {X 0,Y 257.727,Z 519.847,A -85,B 0,C 180,E1 -21026.949,E2 -21026.949} C_VEL
LIN {X 0,Y 258.406,Z 520.448,A -85,B 0,C 180,E1 -21028.283,E2 -21028.283} C_VEL
LIN {X 0,Y 260.033,Z 522.744,A -85,B 0,C 180,E1 -21030.555,E2 -21030.555} C_VEL
LIN {X 0,Y 262.025,Z 526.114,A -85,B 0,C 180,E1 -21032.662,E2 -21032.662} C_VEL
LIN {X 0,Y 263.47,Z 528.916,A -85,B 0,C 180,E1 -21033.961,E2 -21033.961} C_VEL
LIN {X 0,Y 257.91,Z 563.604,A -85,B 0,C 180,E1 -21035.482,E2 -21035.482} C_VEL
LIN {X 0,Y 254.902,Z 577.711,A -85,B 0,C 180,E1 -21036.452,E2 -21036.452} C_VEL
LIN {X 0,Y 251.302,Z 590.552,A -85,B 0,C 180,E1 -21037.641,E2 -21037.641} C_VEL
LIN {X 0,Y 247.404,Z 601.757,A -85,B 0,C 180,E1 -21038.983,E2 -21038.983} C_VEL
LIN {X 0,Y 242.932,Z 612.294,A -85,B 0,C 180,E1 -21040.567,E2 -21040.567} C_VEL
LIN {X 0,Y 238.331,Z 621.889,A -85,B 0,C 180,E1 -21042.407,E2 -21042.407} C_VEL
LIN {X 0,Y 233.249,Z 631.042,A -85,B 0,C 180,E1 -21044.623,E2 -21044.623} C_VEL
LIN {X 0,Y 228.157,Z 638.902,A -85,B 0,C 180,E1 -21047.095,E2 -21047.095} C_VEL
LIN {X 0,Y 223.095,Z 645.953,A -85,B 0,C 180,E1 -21050.022,E2 -21050.022} C_VEL
LIN {X 0,Y 219.176,Z 650.61,A -85,B 0,C 180,E1 -21052.631,E2 -21052.631} C_VEL
LIN {X 0,Y 214.708,Z 655.114,A -85,B 0,C 180,E1 -21056.246,E2 -21056.246} C_VEL
LIN {X 0,Y 212.793,Z 656.718,A -85,B 0,C 180,E1 -21058.107,E2 -21058.107} C_VEL
LIN {X 0,Y 209.927,Z 658.414,A -85,B 0,C 180,E1 -21061.489,E2 -21061.489} C_VEL
LIN {X 0,Y 208.311,Z 658.9,A -85,B 0,C 180,E1 -21063.869,E2 -21063.869} C_VEL
LIN {X 0,Y 207.241,Z 658.811,A -85,B 0,C 180,E1 -21065.839,E2 -21065.839} C_VEL
LIN {X 0,Y 206.132,Z 657.963,A -85,B 0,C 180,E1 -21068.599,E2 -21068.599} C_VEL
LIN {X 0,Y 205.201,Z 655.947,A -85,B 0,C 180,E1 -21071.858,E2 -21071.858} C_VEL
LIN {X 0,Y 204.827,Z 653.014,A -85,B 0,C 180,E1 -21074.912,E2 -21074.912} C_VEL
LIN {X 0,Y 204.744,Z 648.925,A -85,B 0,C 180,E1 -21077.995,E2 -21077.995} C_VEL
LIN {X 0,Y 205.164,Z 642.517,A -85,B 0,C 180,E1 -21081.607,E2 -21081.607} C_VEL
LIN {X 0,Y 205.804,Z 635.406,A -85,B 0,C 180,E1 -21084.729,E2 -21084.729} C_VEL
LIN {X 0,Y 206.755,Z 626.747,A -85,B 0,C 180,E1 -21087.739,E2 -21087.739} C_VEL
LIN {X 0,Y 207.889,Z 617.027,A -85,B 0,C 180,E1 -21090.471,E2 -21090.471} C_VEL
LIN {X 0,Y 209.231,Z 606.262,A -85,B 0,C 180,E1 -21092.886,E2 -21092.886} C_VEL
LIN {X 0,Y 210.456,Z 595.252,A -85,B 0,C 180,E1 -21094.881,E2 -21094.881} C_VEL
LIN {X 0,Y 211.829,Z 582.784,A -85,B 0,C 180,E1 -21096.669,E2 -21096.669} C_VEL
LIN {X 0,Y 213.022,Z 569.18,A -85,B 0,C 180,E1 -21098.164,E2 -21098.164} C_VEL
LIN {X 0,Y 213.988,Z 554.715,A -85,B 0,C 180,E1 -21099.291,E2 -21099.291} C_VEL
LIN {X 0,Y 217.016,Z 492.525,A -85,B 0,C 180,E1 -21102.349,E2 -21102.349} C_VEL
LIN {X 0,Y 217.039,Z 488.296,A -85,B 0,C 180,E1 -21102.565,E2 -21102.565} C_VEL
LIN {X 0,Y 206.712,Z 457.735,A -85,B 0,C 180,E1 -21104.931,E2 -21104.931} C_VEL
LIN {X 0,Y 206.652,Z 457.742,A -85,B 0,C 180,E1 -21109.746,E2 -21109.746} C_VEL
LIN {X 0,Y 206.701,Z 457.735,A -85,B 0,C 180,E1 -21114.688,E2 -21114.688} C_VEL
LIN {X 0,Y 206.697,Z 457.736,A -85,B 0,C 180,E1 -21119.334,E2 -21119.334} C_VEL
LIN {X 0,Y 206.707,Z 457.732,A -85,B 0,C 180,E1 -21123.768,E2 -21123.768} C_VEL
LIN {X 0,Y 206.74,Z 457.732,A -85,B 0,C 180,E1 -21128.04,E2 -21128.04} C_VEL
LIN {X 0,Y 206.875,Z 457.712,A -85,B 0,C 180,E1 -21132.196,E2 -21132.196} C_VEL
LIN {X 0,Y 206.896,Z 457.714,A -85,B 0,C 180,E1 -21136.244,E2 -21136.244} C_VEL
LIN {X 0,Y 207.08,Z 457.687,A -85,B 0,C 180,E1 -21140.229,E2 -21140.229} C_VEL
LIN {X 0,Y 207.047,Z 457.694,A -85,B 0,C 180,E1 -21144.155,E2 -21144.155} C_VEL
LIN {X 0,Y 207.378,Z 457.651,A -85,B 0,C 180,E1 -21148.057,E2 -21148.057} C_VEL
LIN {X 0,Y 207.506,Z 457.633,A -85,B 0,C 180,E1 -21149.999,E2 -21149.999} C_VEL
LIN {X 0,Y 207.377,Z 457.651,A -85,B 0,C 180,E1 -21151.941,E2 -21151.941} C_VEL
LIN {X 0,Y 207.137,Z 457.678,A -85,B 0,C 180,E1 -21157.799,E2 -21157.799} C_VEL
LIN {X 0,Y 206.922,Z 457.708,A -85,B 0,C 180,E1 -21161.758,E2 -21161.758} C_VEL
LIN {X 0,Y 206.846,Z 457.715,A -85,B 0,C 180,E1 -21165.772,E2 -21165.772} C_VEL
LIN {X 0,Y 206.857,Z 457.714,A -85,B 0,C 180,E1 -21167.954,E2 -21167.954} C_VEL
LIN {X 0,Y 206.745,Z 457.728,A -85,B 0,C 180,E1 -21173.39,E2 -21173.39} C_VEL
LIN {X 0,Y 206.688,Z 457.739,A -85,B 0,C 180,E1 -21178.426,E2 -21178.426} C_VEL
LIN {X 0,Y 206.694,Z 457.734,A -85,B 0,C 180,E1 -21182.958,E2 -21182.958} C_VEL
LIN {X 0,Y 206.673,Z 457.739,A -85,B 0,C 180,E1 -21187.741,E2 -21187.741} C_VEL
LIN {X 0,Y 206.633,Z 457.742,A -85,B 0,C 180,E1 -21191.56,E2 -21191.56} C_VEL
LIN {X 0,Y 206.629,Z 457.744,A -85,B 0,C 180,E1 -21195.582,E2 -21195.582} C_VEL
LIN {X 0,Y 206.659,Z 457.739,A -85,B 0,C 180,E1 -21199.748,E2 -21199.748} C_VEL
LIN {X 0,Y 206.698,Z 457.739,A -85,B 0,C 180,E1 -21204.688,E2 -21204.688} C_VEL
LIN {X 0,Y 206.705,Z 457.732,A -85,B 0,C 180,E1 -21209.336,E2 -21209.336} C_VEL
LIN {X 0,Y 206.732,Z 457.732,A -85,B 0,C 180,E1 -21213.772,E2 -21213.772} C_VEL
LIN {X 0,Y 206.757,Z 457.727,A -85,B 0,C 180,E1 -21218.043,E2 -21218.043} C_VEL
LIN {X 0,Y 206.876,Z 457.715,A -85,B 0,C 180,E1 -21222.197,E2 -21222.197} C_VEL
LIN {X 0,Y 206.896,Z 457.711,A -85,B 0,C 180,E1 -21226.244,E2 -21226.244} C_VEL
LIN {X 0,Y 207.105,Z 457.685,A -85,B 0,C 180,E1 -21230.231,E2 -21230.231} C_VEL
LIN {X 0,Y 207.176,Z 457.678,A -85,B 0,C 180,E1 -21232.202,E2 -21232.202} C_VEL
LIN {X 0,Y 207.381,Z 457.649,A -85,B 0,C 180,E1 -21238.058,E2 -21238.058} C_VEL
LIN {X 0,Y 207.514,Z 457.634,A -85,B 0,C 180,E1 -21240,E2 -21240} C_VEL
LIN {X 0,Y 207.382,Z 457.651,A -85,B 0,C 180,E1 -21241.942,E2 -21241.942} C_VEL
LIN {X 0,Y 207.178,Z 457.675,A -85,B 0,C 180,E1 -21247.799,E2 -21247.799} C_VEL
LIN {X 0,Y 206.983,Z 457.699,A -85,B 0,C 180,E1 -21251.755,E2 -21251.755} C_VEL
LIN {X 0,Y 206.867,Z 457.714,A -85,B 0,C 180,E1 -21255.771,E2 -21255.771} C_VEL
LIN {X 0,Y 206.778,Z 457.726,A -85,B 0,C 180,E1 -21259.87,E2 -21259.87} C_VEL
LIN {X 0,Y 206.747,Z 457.728,A -85,B 0,C 180,E1 -21264.074,E2 -21264.074} C_VEL
LIN {X 0,Y 206.744,Z 457.732,A -85,B 0,C 180,E1 -21268.419,E2 -21268.419} C_VEL
LIN {X 0,Y 206.702,Z 457.737,A -85,B 0,C 180,E1 -21272.957,E2 -21272.957} C_VEL
LIN {X 0,Y 206.679,Z 457.737,A -85,B 0,C 180,E1 -21277.74,E2 -21277.74} C_VEL
LIN {X 0,Y 206.642,Z 457.741,A -85,B 0,C 180,E1 -21281.564,E2 -21281.564} C_VEL
LIN {X 0,Y 206.635,Z 457.743,A -85,B 0,C 180,E1 -21285.582,E2 -21285.582} C_VEL
LIN {X 0,Y 206.678,Z 457.736,A -85,B 0,C 180,E1 -21289.754,E2 -21289.754} C_VEL
LIN {X 0,Y 206.828,Z 457.889,A -85,B 0,C 180,E1 -21292.077,E2 -21292.077} C_VEL
LIN {X 0,Y 209.151,Z 469.566,A -85,B 0,C 180,E1 -21296.728,E2 -21296.728} C_VEL
LIN {X 0,Y 210.684,Z 476.923,A -85,B 0,C 180,E1 -21299.554,E2 -21299.554} C_VEL
LIN {X 0,Y 212.068,Z 482.762,A -85,B 0,C 180,E1 -21299.971,E2 -21299.971} C_VEL
LIN {X 0,Y 213.97,Z 512.695,A -85,B 0,C 180,E1 -21301.662,E2 -21301.662} C_VEL
LIN {X 0,Y 216.088,Z 538.4,A -85,B 0,C 180,E1 -21303.11,E2 -21303.11} C_VEL
LIN {X 0,Y 216.01,Z 539.554,A -85,B 0,C 180,E1 -21303.165,E2 -21303.165} C_VEL
LIN {X 0,Y 215.11,Z 545.317,A -85,B 0,C 180,E1 -21303.415,E2 -21303.415} C_VEL
LIN {X 0,Y 208.475,Z 563.884,A -85,B 0,C 180,E1 -21304.063,E2 -21304.063} C_VEL
LIN {X 0,Y 207.534,Z 569.646,A -85,B 0,C 180,E1 -21304.329,E2 -21304.329} C_VEL
LIN {X 0,Y 206.492,Z 589.13,A -85,B 0,C 180,E1 -21305.427,E2 -21305.427} C_VEL
LIN {X 0,Y 205.468,Z 602.478,A -85,B 0,C 180,E1 -21306.571,E2 -21306.571} C_VEL
LIN {X 0,Y 203.935,Z 616.224,A -85,B 0,C 180,E1 -21308.196,E2 -21308.196} C_VEL
LIN {X 0,Y 202.447,Z 628.982,A -85,B 0,C 180,E1 -21310.217,E2 -21310.217} C_VEL
LIN {X 0,Y 201.122,Z 640.138,A -85,B 0,C 180,E1 -21312.46,E2 -21312.46} C_VEL
LIN {X 0,Y 199.994,Z 649.163,A -85,B 0,C 180,E1 -21314.719,E2 -21314.719} C_VEL
LIN {X 0,Y 199.04,Z 658.987,A -85,B 0,C 180,E1 -21317.77,E2 -21317.77} C_VEL
LIN {X 0,Y 198.578,Z 666.791,A -85,B 0,C 180,E1 -21320.837,E2 -21320.837} C_VEL
LIN {X 0,Y 198.44,Z 672.958,A -85,B 0,C 180,E1 -21323.902,E2 -21323.902} C_VEL
LIN {X 0,Y 198.522,Z 677.725,A -85,B 0,C 180,E1 -21326.957,E2 -21326.957} C_VEL
LIN {X 0,Y 198.57,Z 681.207,A -85,B 0,C 180,E1 -21330.001,E2 -21330.001} C_VEL
LIN {X 0,Y 198.262,Z 682.857,A -85,B 0,C 180,E1 -21332.032,E2 -21332.032} C_VEL
LIN {X 0,Y 197.786,Z 684.661,A -85,B 0,C 180,E1 -21335.768,E2 -21335.768} C_VEL
LIN {X 0,Y 197.724,Z 685.082,A -85,B 0,C 180,E1 -21338.175,E2 -21338.175} C_VEL
LIN {X 0,Y 198.416,Z 684.637,A -85,B 0,C 180,E1 -21342.271,E2 -21342.271} C_VEL
LIN {X 0,Y 199.136,Z 683.849,A -85,B 0,C 180,E1 -21344.304,E2 -21344.304} C_VEL
LIN {X 0,Y 201.605,Z 681.113,A -85,B 0,C 180,E1 -21348.286,E2 -21348.286} C_VEL
LIN {X 0,Y 205.121,Z 676.837,A -85,B 0,C 180,E1 -21352.142,E2 -21352.142} C_VEL
LIN {X 0,Y 208.479,Z 672.532,A -85,B 0,C 180,E1 -21354.923,E2 -21354.923} C_VEL
LIN {X 0,Y 213.196,Z 666.187,A -85,B 0,C 180,E1 -21358.019,E2 -21358.019} C_VEL
LIN {X 0,Y 218.761,Z 658.228,A -85,B 0,C 180,E1 -21360.933,E2 -21360.933} C_VEL
LIN {X 0,Y 224.138,Z 649.858,A -85,B 0,C 180,E1 -21363.28,E2 -21363.28} C_VEL
LIN {X 0,Y 230.002,Z 639.737,A -85,B 0,C 180,E1 -21365.491,E2 -21365.491} C_VEL
LIN {X 0,Y 235.918,Z 628.405,A -85,B 0,C 180,E1 -21367.372,E2 -21367.372} C_VEL
LIN {X 0,Y 241.143,Z 616.993,A -85,B 0,C 180,E1 -21368.801,E2 -21368.801} C_VEL
LIN {X 0,Y 246.584,Z 602.791,A -85,B 0,C 180,E1 -21370.155,E2 -21370.155} C_VEL
LIN {X 0,Y 250.313,Z 590.816,A -85,B 0,C 180,E1 -21371.019,E2 -21371.019} C_VEL
LIN {X 0,Y 253.991,Z 575.518,A -85,B 0,C 180,E1 -21371.811,E2 -21371.811} C_VEL
LIN {X 0,Y 258.243,Z 549.315,A -85,B 0,C 180,E1 -21372.94,E2 -21372.94} C_VEL
LIN {X 0,Y 258.697,Z 543.32,A -85,B 0,C 180,E1 -21373.552,E2 -21373.552} C_VEL
LIN {X 0,Y 257.511,Z 538.227,A -85,B 0,C 180,E1 -21375.249,E2 -21375.249} C_VEL
LIN {X 0,Y 256.667,Z 534.771,A -85,B 0,C 180,E1 -21376.733,E2 -21376.733} C_VEL
LIN {X 0,Y 255.851,Z 531.118,A -85,B 0,C 180,E1 -21378.634,E2 -21378.634} C_VEL
LIN {X 0,Y 255.143,Z 527.79,A -85,B 0,C 180,E1 -21381.791,E2 -21381.791} C_VEL
LIN {X 0,Y 255.231,Z 526.663,A -85,B 0,C 180,E1 -21383.914,E2 -21383.914} C_VEL
LIN {X 0,Y 256.385,Z 526.816,A -85,B 0,C 180,E1 -21387.349,E2 -21387.349} C_VEL
LIN {X 0,Y 258.092,Z 529.307,A -85,B 0,C 180,E1 -21390.123,E2 -21390.123} C_VEL
LIN {X 0,Y 259.91,Z 532.564,A -85,B 0,C 180,E1 -21392.216,E2 -21392.216} C_VEL
LIN {X 0,Y 260.348,Z 533.496,A -85,B 0,C 180,E1 -21392.683,E2 -21392.683} C_VEL
LIN {X 0,Y 255.028,Z 564.783,A -85,B 0,C 180,E1 -21394.057,E2 -21394.057} C_VEL
LIN {X 0,Y 252.124,Z 577.867,A -85,B 0,C 180,E1 -21394.953,E2 -21394.953} C_VEL
LIN {X 0,Y 248.682,Z 589.599,A -85,B 0,C 180,E1 -21396.004,E2 -21396.004} C_VEL
LIN {X 0,Y 244.007,Z 602.309,A -85,B 0,C 180,E1 -21397.501,E2 -21397.501} C_VEL
LIN {X 0,Y 239.264,Z 613.09,A -85,B 0,C 180,E1 -21399.113,E2 -21399.113} C_VEL
LIN {X 0,Y 234.727,Z 621.885,A -85,B 0,C 180,E1 -21400.77,E2 -21400.77} C_VEL
LIN {X 0,Y 228.969,Z 631.664,A -85,B 0,C 180,E1 -21403.139,E2 -21403.139} C_VEL
LIN {X 0,Y 223.894,Z 639.11,A -85,B 0,C 180,E1 -21405.456,E2 -21405.456} C_VEL
LIN {X 0,Y 219.143,Z 645.276,A -85,B 0,C 180,E1 -21407.968,E2 -21407.968} C_VEL
LIN {X 0,Y 214.805,Z 650.228,A -85,B 0,C 180,E1 -21410.585,E2 -21410.585} C_VEL
LIN {X 0,Y 210.953,Z 654.054,A -85,B 0,C 180,E1 -21413.304,E2 -21413.304} C_VEL
LIN {X 0,Y 207.588,Z 656.822,A -85,B 0,C 180,E1 -21416.117,E2 -21416.117} C_VEL
LIN {X 0,Y 205.619,Z 658.141,A -85,B 0,C 180,E1 -21418.041,E2 -21418.041} C_VEL
LIN {X 0,Y 203.04,Z 659.304,A -85,B 0,C 180,E1 -21421.094,E2 -21421.094} C_VEL
LIN {X 0,Y 201.084,Z 659.564,A -85,B 0,C 180,E1 -21424.008,E2 -21424.008} C_VEL
LIN {X 0,Y 200.006,Z 659.222,A -85,B 0,C 180,E1 -21426.051,E2 -21426.051} C_VEL
LIN {X 0,Y 199.01,Z 658.207,A -85,B 0,C 180,E1 -21428.573,E2 -21428.573} C_VEL
LIN {X 0,Y 198.009,Z 655.581,A -85,B 0,C 180,E1 -21432.296,E2 -21432.296} C_VEL
LIN {X 0,Y 197.724,Z 652.406,A -85,B 0,C 180,E1 -21435.319,E2 -21435.319} C_VEL
LIN {X 0,Y 197.707,Z 647.731,A -85,B 0,C 180,E1 -21438.658,E2 -21438.658} C_VEL
LIN {X 0,Y 198.096,Z 641.984,A -85,B 0,C 180,E1 -21441.826,E2 -21441.826} C_VEL
LIN {X 0,Y 198.811,Z 634.402,A -85,B 0,C 180,E1 -21445.1,E2 -21445.1} C_VEL
LIN {X 0,Y 199.685,Z 626.462,A -85,B 0,C 180,E1 -21447.875,E2 -21447.875} C_VEL
LIN {X 0,Y 200.776,Z 617.3,A -85,B 0,C 180,E1 -21450.501,E2 -21450.501} C_VEL
LIN {X 0,Y 202.187,Z 605.957,A -85,B 0,C 180,E1 -21453.111,E2 -21453.111} C_VEL
LIN {X 0,Y 203.588,Z 593.898,A -85,B 0,C 180,E1 -21455.325,E2 -21455.325} C_VEL
LIN {X 0,Y 204.972,Z 580.944,A -85,B 0,C 180,E1 -21457.18,E2 -21457.18} C_VEL
LIN {X 0,Y 206.083,Z 568.205,A -85,B 0,C 180,E1 -21458.573,E2 -21458.573} C_VEL
LIN {X 0,Y 207.019,Z 554.721,A -85,B 0,C 180,E1 -21459.637,E2 -21459.637} C_VEL
LIN {X 0,Y 210.263,Z 490.025,A -85,B 0,C 180,E1 -21462.927,E2 -21462.927} C_VEL
LIN {X 0,Y 199.636,Z 458.615,A -85,B 0,C 180,E1 -21465.453,E2 -21465.453} C_VEL
LIN {X 0,Y 199.598,Z 458.621,A -85,B 0,C 180,E1 -21470.772,E2 -21470.772} C_VEL
LIN {X 0,Y 199.612,Z 458.617,A -85,B 0,C 180,E1 -21475.712,E2 -21475.712} C_VEL
LIN {X 0,Y 199.687,Z 458.611,A -85,B 0,C 180,E1 -21478.134,E2 -21478.134} C_VEL
LIN {X 0,Y 199.645,Z 458.613,A -85,B 0,C 180,E1 -21482.765,E2 -21482.765} C_VEL
LIN {X 0,Y 199.712,Z 458.606,A -85,B 0,C 180,E1 -21487.225,E2 -21487.225} C_VEL
LIN {X 0,Y 199.798,Z 458.591,A -85,B 0,C 180,E1 -21491.757,E2 -21491.757} C_VEL
LIN {X 0,Y 199.837,Z 458.591,A -85,B 0,C 180,E1 -21495.748,E2 -21495.748} C_VEL
LIN {X 0,Y 200.024,Z 458.565,A -85,B 0,C 180,E1 -21499.881,E2 -21499.881} C_VEL
LIN {X 0,Y 200.009,Z 458.57,A -85,B 0,C 180,E1 -21503.948,E2 -21503.948} C_VEL
LIN {X 0,Y 200.317,Z 458.53,A -85,B 0,C 180,E1 -21507.989,E2 -21507.989} C_VEL
LIN {X 0,Y 200.471,Z 458.509,A -85,B 0,C 180,E1 -21509.999,E2 -21509.999} C_VEL
LIN {X 0,Y 200.016,Z 458.569,A -85,B 0,C 180,E1 -21514.029,E2 -21514.029} C_VEL
LIN {X 0,Y 200.087,Z 458.557,A -85,B 0,C 180,E1 -21518.076,E2 -21518.076} C_VEL
LIN {X 0,Y 199.871,Z 458.588,A -85,B 0,C 180,E1 -21522.179,E2 -21522.179} C_VEL
LIN {X 0,Y 199.789,Z 458.595,A -85,B 0,C 180,E1 -21526.344,E2 -21526.344} C_VEL
LIN {X 0,Y 199.674,Z 458.614,A -85,B 0,C 180,E1 -21530.607,E2 -21530.607} C_VEL
LIN {X 0,Y 199.65,Z 458.611,A -85,B 0,C 180,E1 -21534.987,E2 -21534.987} C_VEL
LIN {X 0,Y 199.608,Z 458.619,A -85,B 0,C 180,E1 -21539.532,E2 -21539.532} C_VEL
LIN {X 0,Y 199.665,Z 458.614,A -85,B 0,C 180,E1 -21542.352,E2 -21542.352} C_VEL
LIN {X 0,Y 199.619,Z 458.62,A -85,B 0,C 180,E1 -21546.763,E2 -21546.763} C_VEL
LIN {X 0,Y 199.596,Z 458.621,A -85,B 0,C 180,E1 -21549.33,E2 -21549.33} C_VEL
LIN {X 0,Y 199.567,Z 458.623,A -85,B 0,C 180,E1 -21552.308,E2 -21552.308} C_VEL
LIN {X 0,Y 199.576,Z 458.623,A -85,B 0,C 180,E1 -21555.227,E2 -21555.227} C_VEL
LIN {X 0,Y 199.576,Z 458.624,A -85,B 0,C 180,E1 -21558.004,E2 -21558.004} C_VEL
LIN {X 0,Y 199.609,Z 458.617,A -85,B 0,C 180,E1 -21560.767,E2 -21560.767} C_VEL
LIN {X 0,Y 199.61,Z 458.619,A -85,B 0,C 180,E1 -21565.713,E2 -21565.713} C_VEL
LIN {X 0,Y 199.692,Z 458.609,A -85,B 0,C 180,E1 -21568.135,E2 -21568.135} C_VEL
LIN {X 0,Y 199.685,Z 458.612,A -85,B 0,C 180,E1 -21572.772,E2 -21572.772} C_VEL
LIN {X 0,Y 199.737,Z 458.601,A -85,B 0,C 180,E1 -21577.229,E2 -21577.229} C_VEL
LIN {X 0,Y 199.837,Z 458.59,A -85,B 0,C 180,E1 -21581.722,E2 -21581.722} C_VEL
LIN {X 0,Y 199.836,Z 458.589,A -85,B 0,C 180,E1 -21585.748,E2 -21585.748} C_VEL
LIN {X 0,Y 200.069,Z 458.561,A -85,B 0,C 180,E1 -21589.884,E2 -21589.884} C_VEL
LIN {X 0,Y 200.034,Z 458.566,A -85,B 0,C 180,E1 -21593.95,E2 -21593.95} C_VEL
LIN {X 0,Y 200.32,Z 458.529,A -85,B 0,C 180,E1 -21597.99,E2 -21597.99} C_VEL
LIN {X 0,Y 200.479,Z 458.511,A -85,B 0,C 180,E1 -21600,E2 -21600} C_VEL
LIN {X 0,Y 200.031,Z 458.565,A -85,B 0,C 180,E1 -21604.03,E2 -21604.03} C_VEL
LIN {X 0,Y 200.124,Z 458.555,A -85,B 0,C 180,E1 -21608.075,E2 -21608.075} C_VEL
LIN {X 0,Y 199.914,Z 458.581,A -85,B 0,C 180,E1 -21612.177,E2 -21612.177} C_VEL
LIN {X 0,Y 199.804,Z 458.595,A -85,B 0,C 180,E1 -21616.344,E2 -21616.344} C_VEL
LIN {X 0,Y 199.69,Z 458.61,A -85,B 0,C 180,E1 -21620.607,E2 -21620.607} C_VEL
LIN {X 0,Y 199.664,Z 458.614,A -85,B 0,C 180,E1 -21624.986,E2 -21624.986} C_VEL
LIN {X 0,Y 199.674,Z 458.609,A -85,B 0,C 180,E1 -21629.523,E2 -21629.523} C_VEL
LIN {X 0,Y 199.677,Z 458.608,A -85,B 0,C 180,E1 -21632.359,E2 -21632.359} C_VEL
LIN {X 0,Y 199.623,Z 458.62,A -85,B 0,C 180,E1 -21636.764,E2 -21636.764} C_VEL
LIN {X 0,Y 199.608,Z 458.616,A -85,B 0,C 180,E1 -21639.329,E2 -21639.329} C_VEL
LIN {X 0,Y 199.575,Z 458.623,A -85,B 0,C 180,E1 -21642.311,E2 -21642.311} C_VEL
LIN {X 0,Y 199.581,Z 458.623,A -85,B 0,C 180,E1 -21645.23,E2 -21645.23} C_VEL
LIN {X 0,Y 199.679,Z 458.611,A -85,B 0,C 180,E1 -21650.744,E2 -21650.744} C_VEL
LIN {X 0,Y 199.792,Z 458.8,A -85,B 0,C 180,E1 -21651.814,E2 -21651.814} C_VEL
LIN {X 0,Y 202.099,Z 470.37,A -85,B 0,C 180,E1 -21656.575,E2 -21656.575} C_VEL
LIN {X 0,Y 203.352,Z 476.555,A -85,B 0,C 180,E1 -21658.991,E2 -21658.991} C_VEL
LIN {X 0,Y 205.224,Z 484.193,A -85,B 0,C 180,E1 -21659.554,E2 -21659.554} C_VEL
LIN {X 0,Y 207.13,Z 513.991,A -85,B 0,C 180,E1 -21661.314,E2 -21661.314} C_VEL
LIN {X 0,Y 209.109,Z 538.568,A -85,B 0,C 180,E1 -21662.747,E2 -21662.747} C_VEL
LIN {X 0,Y 207.534,Z 569.646,A -85,B 0,C 180,E1 -21664.329,E2 -21664.329} C_VEL
LIN {X 0,Y 206.578,Z 575.396,A -85,B 0,C 180,E1 -21664.59,E2 -21664.59} C_VEL
LIN {X 0,Y 203.205,Z 584.62,A -85,B 0,C 180,E1 -21664.98,E2 -21664.98} C_VEL
LIN {X 0,Y 199.772,Z 593.73,A -85,B 0,C 180,E1 -21665.545,E2 -21665.545} C_VEL
LIN {X 0,Y 198.69,Z 599.302,A -85,B 0,C 180,E1 -21666.042,E2 -21666.042} C_VEL
LIN {X 0,Y 197.326,Z 611.761,A -85,B 0,C 180,E1 -21667.47,E2 -21667.47} C_VEL
LIN {X 0,Y 195.78,Z 625.154,A -85,B 0,C 180,E1 -21669.513,E2 -21669.513} C_VEL
LIN {X 0,Y 194.365,Z 636.84,A -85,B 0,C 180,E1 -21671.829,E2 -21671.829} C_VEL
LIN {X 0,Y 193.148,Z 646.324,A -85,B 0,C 180,E1 -21674.164,E2 -21674.164} C_VEL
LIN {X 0,Y 192.275,Z 655.086,A -85,B 0,C 180,E1 -21676.795,E2 -21676.795} C_VEL
LIN {X 0,Y 191.655,Z 663.546,A -85,B 0,C 180,E1 -21679.97,E2 -21679.97} C_VEL
LIN {X 0,Y 191.456,Z 670.329,A -85,B 0,C 180,E1 -21683.167,E2 -21683.167} C_VEL
LIN {X 0,Y 191.474,Z 674.755,A -85,B 0,C 180,E1 -21685.791,E2 -21685.791} C_VEL
LIN {X 0,Y 191.578,Z 678.874,A -85,B 0,C 180,E1 -21688.95,E2 -21688.95} C_VEL
LIN {X 0,Y 191.567,Z 679.967,A -85,B 0,C 180,E1 -21690.001,E2 -21690.001} C_VEL
LIN {X 0,Y 191.239,Z 681.694,A -85,B 0,C 180,E1 -21692.107,E2 -21692.107} C_VEL
LIN {X 0,Y 190.693,Z 683.856,A -85,B 0,C 180,E1 -21696.349,E2 -21696.349} C_VEL
LIN {X 0,Y 190.679,Z 684.331,A -85,B 0,C 180,E1 -21698.479,E2 -21698.479} C_VEL
LIN {X 0,Y 191.462,Z 684.106,A -85,B 0,C 180,E1 -21702.724,E2 -21702.724} C_VEL
LIN {X 0,Y 192.232,Z 683.444,A -85,B 0,C 180,E1 -21704.829,E2 -21704.829} C_VEL
LIN {X 0,Y 194.845,Z 681.035,A -85,B 0,C 180,E1 -21708.944,E2 -21708.944} C_VEL
LIN {X 0,Y 198.556,Z 677.074,A -85,B 0,C 180,E1 -21712.915,E2 -21712.915} C_VEL
LIN {X 0,Y 203.436,Z 671.477,A -85,B 0,C 180,E1 -21716.687,E2 -21716.687} C_VEL
LIN {X 0,Y 208.584,Z 665.127,A -85,B 0,C 180,E1 -21719.802,E2 -21719.802} C_VEL
LIN {X 0,Y 214.613,Z 657.072,A -85,B 0,C 180,E1 -21722.707,E2 -21722.707} C_VEL
LIN {X 0,Y 220.358,Z 648.739,A -85,B 0,C 180,E1 -21725.036,E2 -21725.036} C_VEL
LIN {X 0,Y 225.505,Z 640.442,A -85,B 0,C 180,E1 -21726.866,E2 -21726.866} C_VEL
LIN {X 0,Y 231.659,Z 629.423,A -85,B 0,C 180,E1 -21728.736,E2 -21728.736} C_VEL
LIN {X 0,Y 237.699,Z 617.227,A -85,B 0,C 180,E1 -21730.3,E2 -21730.3} C_VEL
LIN {X 0,Y 242.712,Z 605.093,A -85,B 0,C 180,E1 -21731.482,E2 -21731.482} C_VEL
LIN {X 0,Y 246.56,Z 593.85,A -85,B 0,C 180,E1 -21732.332,E2 -21732.332} C_VEL
LIN {X 0,Y 250.603,Z 579.204,A -85,B 0,C 180,E1 -21733.148,E2 -21733.148} C_VEL
LIN {X 0,Y 254.713,Z 557.052,A -85,B 0,C 180,E1 -21734.109,E2 -21734.109} C_VEL
LIN {X 0,Y 255.806,Z 550.339,A -85,B 0,C 180,E1 -21734.436,E2 -21734.436} C_VEL
LIN {X 0,Y 256.013,Z 547.574,A -85,B 0,C 180,E1 -21734.754,E2 -21734.754} C_VEL
LIN {X 0,Y 254.889,Z 541.923,A -85,B 0,C 180,E1 -21736.875,E2 -21736.875} C_VEL
LIN {X 0,Y 254.045,Z 537.6,A -85,B 0,C 180,E1 -21739.163,E2 -21739.163} C_VEL
LIN {X 0,Y 253.546,Z 534.442,A -85,B 0,C 180,E1 -21742.264,E2 -21742.264} C_VEL
LIN {X 0,Y 253.687,Z 533.565,A -85,B 0,C 180,E1 -21744.006,E2 -21744.006} C_VEL
LIN {X 0,Y 254.78,Z 533.707,A -85,B 0,C 180,E1 -21747.27,E2 -21747.27} C_VEL
LIN {X 0,Y 256.201,Z 535.896,A -85,B 0,C 180,E1 -21749.727,E2 -21749.727} C_VEL
LIN {X 0,Y 257.426,Z 538.281,A -85,B 0,C 180,E1 -21751.348,E2 -21751.348} C_VEL
LIN {X 0,Y 252.416,Z 566.323,A -85,B 0,C 180,E1 -21752.61,E2 -21752.61} C_VEL
LIN {X 0,Y 249.218,Z 579.473,A -85,B 0,C 180,E1 -21753.518,E2 -21753.518} C_VEL
LIN {X 0,Y 244.985,Z 592.677,A -85,B 0,C 180,E1 -21754.74,E2 -21754.74} C_VEL
LIN {X 0,Y 240.164,Z 604.819,A -85,B 0,C 180,E1 -21756.208,E2 -21756.208} C_VEL
LIN {X 0,Y 234.774,Z 615.877,A -85,B 0,C 180,E1 -21757.933,E2 -21757.933} C_VEL
LIN {X 0,Y 229.411,Z 625.412,A -85,B 0,C 180,E1 -21759.84,E2 -21759.84} C_VEL
LIN {X 0,Y 223.568,Z 634.341,A -85,B 0,C 180,E1 -21762.152,E2 -21762.152} C_VEL
LIN {X 0,Y 217.185,Z 642.674,A -85,B 0,C 180,E1 -21764.996,E2 -21764.996} C_VEL
LIN {X 0,Y 212.321,Z 648.283,A -85,B 0,C 180,E1 -21767.575,E2 -21767.575} C_VEL
LIN {X 0,Y 207.844,Z 652.703,A -85,B 0,C 180,E1 -21770.266,E2 -21770.266} C_VEL
LIN {X 0,Y 205.138,Z 655.05,A -85,B 0,C 180,E1 -21772.123,E2 -21772.123} C_VEL
LIN {X 0,Y 202.702,Z 656.969,A -85,B 0,C 180,E1 -21774.029,E2 -21774.029} C_VEL
LIN {X 0,Y 200.441,Z 658.416,A -85,B 0,C 180,E1 -21775.979,E2 -21775.979} C_VEL
LIN {X 0,Y 196.685,Z 660.07,A -85,B 0,C 180,E1 -21780,E2 -21780} C_VEL
LIN {X 0,Y 195.151,Z 660.301,A -85,B 0,C 180,E1 -21782.064,E2 -21782.064} C_VEL
LIN {X 0,Y 193.845,Z 660.088,A -85,B 0,C 180,E1 -21784.158,E2 -21784.158} C_VEL
LIN {X 0,Y 191.957,Z 658.453,A -85,B 0,C 180,E1 -21788.421,E2 -21788.421} C_VEL
LIN {X 0,Y 191.278,Z 656.995,A -85,B 0,C 180,E1 -21790.586,E2 -21790.586} C_VEL
LIN {X 0,Y 190.719,Z 653.95,A -85,B 0,C 180,E1 -21793.858,E2 -21793.858} C_VEL
LIN {X 0,Y 190.553,Z 649.771,A -85,B 0,C 180,E1 -21797.161,E2 -21797.161} C_VEL
LIN {X 0,Y 190.896,Z 643.301,A -85,B 0,C 180,E1 -21801.036,E2 -21801.036} C_VEL
LIN {X 0,Y 191.513,Z 636.122,A -85,B 0,C 180,E1 -21804.383,E2 -21804.383} C_VEL
LIN {X 0,Y 192.343,Z 628.707,A -85,B 0,C 180,E1 -21807.177,E2 -21807.177} C_VEL
LIN {X 0,Y 193.488,Z 619.071,A -85,B 0,C 180,E1 -21810.12,E2 -21810.12} C_VEL
LIN {X 0,Y 194.821,Z 608.371,A -85,B 0,C 180,E1 -21812.759,E2 -21812.759} C_VEL
LIN {X 0,Y 196.152,Z 597.163,A -85,B 0,C 180,E1 -21814.978,E2 -21814.978} C_VEL
LIN {X 0,Y 197.524,Z 585.02,A -85,B 0,C 180,E1 -21816.9,E2 -21816.9} C_VEL
LIN {X 0,Y 198.783,Z 571.401,A -85,B 0,C 180,E1 -21818.545,E2 -21818.545} C_VEL
LIN {X 0,Y 199.838,Z 558.072,A -85,B 0,C 180,E1 -21819.723,E2 -21819.723} C_VEL
LIN {X 0,Y 200.82,Z 537.393,A -85,B 0,C 180,E1 -21820.926,E2 -21820.926} C_VEL
LIN {X 0,Y 203.281,Z 491.234,A -85,B 0,C 180,E1 -21823.345,E2 -21823.345} C_VEL
LIN {X 0,Y 192.599,Z 459.492,A -85,B 0,C 180,E1 -21826.015,E2 -21826.015} C_VEL
LIN {X 0,Y 192.543,Z 459.499,A -85,B 0,C 180,E1 -21831.645,E2 -21831.645} C_VEL
LIN {X 0,Y 192.596,Z 459.494,A -85,B 0,C 180,E1 -21836.813,E2 -21836.813} C_VEL
LIN {X 0,Y 192.622,Z 459.487,A -85,B 0,C 180,E1 -21841.684,E2 -21841.684} C_VEL
LIN {X 0,Y 192.681,Z 459.484,A -85,B 0,C 180,E1 -21846.344,E2 -21846.344} C_VEL
LIN {X 0,Y 192.734,Z 459.471,A -85,B 0,C 180,E1 -21851.457,E2 -21851.457} C_VEL
LIN {X 0,Y 192.765,Z 459.472,A -85,B 0,C 180,E1 -21855.213,E2 -21855.213} C_VEL
LIN {X 0,Y 192.947,Z 459.446,A -85,B 0,C 180,E1 -21859.566,E2 -21859.566} C_VEL
LIN {X 0,Y 192.973,Z 459.446,A -85,B 0,C 180,E1 -21863.727,E2 -21863.727} C_VEL
LIN {X 0,Y 193.259,Z 459.409,A -85,B 0,C 180,E1 -21867.915,E2 -21867.915} C_VEL
LIN {X 0,Y 193.436,Z 459.385,A -85,B 0,C 180,E1 -21869.999,E2 -21869.999} C_VEL
LIN {X 0,Y 192.962,Z 459.449,A -85,B 0,C 180,E1 -21874.177,E2 -21874.177} C_VEL
LIN {X 0,Y 193.035,Z 459.436,A -85,B 0,C 180,E1 -21878.373,E2 -21878.373} C_VEL
LIN {X 0,Y 192.797,Z 459.47,A -85,B 0,C 180,E1 -21882.633,E2 -21882.633} C_VEL
LIN {X 0,Y 192.748,Z 459.472,A -85,B 0,C 180,E1 -21886.959,E2 -21886.959} C_VEL
LIN {X 0,Y 192.609,Z 459.491,A -85,B 0,C 180,E1 -21891.4,E2 -21891.4} C_VEL
LIN {X 0,Y 192.639,Z 459.487,A -85,B 0,C 180,E1 -21894.207,E2 -21894.207} C_VEL
LIN {X 0,Y 192.601,Z 459.494,A -85,B 0,C 180,E1 -21898.865,E2 -21898.865} C_VEL
LIN {X 0,Y 192.594,Z 459.489,A -85,B 0,C 180,E1 -21903.186,E2 -21903.186} C_VEL
LIN {X 0,Y 192.543,Z 459.502,A -85,B 0,C 180,E1 -21908.353,E2 -21908.353} C_VEL
LIN {X 0,Y 192.485,Z 459.504,A -85,B 0,C 180,E1 -21913.094,E2 -21913.094} C_VEL
LIN {X 0,Y 192.488,Z 459.508,A -85,B 0,C 180,E1 -21916.904,E2 -21916.904} C_VEL
LIN {X 0,Y 192.55,Z 459.494,A -85,B 0,C 180,E1 -21921.648,E2 -21921.648} C_VEL
LIN {X 0,Y 192.595,Z 459.494,A -85,B 0,C 180,E1 -21926.814,E2 -21926.814} C_VEL
LIN {X 0,Y 192.66,Z 459.483,A -85,B 0,C 180,E1 -21931.691,E2 -21931.691} C_VEL
LIN {X 0,Y 192.705,Z 459.481,A -85,B 0,C 180,E1 -21936.349,E2 -21936.349} C_VEL
LIN {X 0,Y 192.78,Z 459.469,A -85,B 0,C 180,E1 -21941.414,E2 -21941.414} C_VEL
LIN {X 0,Y 192.764,Z 459.471,A -85,B 0,C 180,E1 -21945.214,E2 -21945.214} C_VEL
LIN {X 0,Y 192.98,Z 459.444,A -85,B 0,C 180,E1 -21949.509,E2 -21949.509} C_VEL
LIN {X 0,Y 193.067,Z 459.434,A -85,B 0,C 180,E1 -21951.628,E2 -21951.628} C_VEL
LIN {X 0,Y 193.262,Z 459.408,A -85,B 0,C 180,E1 -21957.916,E2 -21957.916} C_VEL
LIN {X 0,Y 193.443,Z 459.387,A -85,B 0,C 180,E1 -21960,E2 -21960} C_VEL
LIN {X 0,Y 192.978,Z 459.444,A -85,B 0,C 180,E1 -21964.177,E2 -21964.177} C_VEL
LIN {X 0,Y 193.072,Z 459.434,A -85,B 0,C 180,E1 -21968.372,E2 -21968.372} C_VEL
LIN {X 0,Y 192.853,Z 459.46,A -85,B 0,C 180,E1 -21972.63,E2 -21972.63} C_VEL
LIN {X 0,Y 192.757,Z 459.475,A -85,B 0,C 180,E1 -21976.959,E2 -21976.959} C_VEL
LIN {X 0,Y 192.621,Z 459.487,A -85,B 0,C 180,E1 -21981.399,E2 -21981.399} C_VEL
LIN {X 0,Y 192.647,Z 459.485,A -85,B 0,C 180,E1 -21984.214,E2 -21984.214} C_VEL
LIN {X 0,Y 192.65,Z 459.486,A -85,B 0,C 180,E1 -21988.893,E2 -21988.893} C_VEL
LIN {X 0,Y 192.598,Z 459.493,A -85,B 0,C 180,E1 -21993.186,E2 -21993.186} C_VEL
LIN {X 0,Y 192.551,Z 459.499,A -85,B 0,C 180,E1 -21998.352,E2 -21998.352} C_VEL
LIN {X 0,Y 192.492,Z 459.507,A -85,B 0,C 180,E1 -22003.097,E2 -22003.097} C_VEL
LIN {X 0,Y 192.492,Z 459.505,A -85,B 0,C 180,E1 -22006.905,E2 -22006.905} C_VEL
LIN {X 0,Y 192.721,Z 459.679,A -85,B 0,C 180,E1 -22011.536,E2 -22011.536} C_VEL
LIN {X 0,Y 194.843,Z 470.276,A -85,B 0,C 180,E1 -22016.059,E2 -22016.059} C_VEL
LIN {X 0,Y 196.03,Z 475.978,A -85,B 0,C 180,E1 -22018.397,E2 -22018.397} C_VEL
LIN {X 0,Y 198.397,Z 485.681,A -85,B 0,C 180,E1 -22019.136,E2 -22019.136} C_VEL
LIN {X 0,Y 200.42,Z 517.165,A -85,B 0,C 180,E1 -22021.057,E2 -22021.057} C_VEL
LIN {X 0,Y 202.129,Z 538.887,A -85,B 0,C 180,E1 -22022.377,E2 -22022.377} C_VEL
LIN {X 0,Y 199.696,Z 586.227,A -85,B 0,C 180,E1 -22024.95,E2 -22024.95} C_VEL
LIN {X 0,Y 198.69,Z 599.302,A -85,B 0,C 180,E1 -22026.042,E2 -22026.042} C_VEL
LIN {X 0,Y 197.466,Z 604.764,A -85,B 0,C 180,E1 -22026.589,E2 -22026.589} C_VEL
LIN {X 0,Y 193.682,Z 613.262,A -85,B 0,C 180,E1 -22027.596,E2 -22027.596} C_VEL
LIN {X 0,Y 189.822,Z 621.434,A -85,B 0,C 180,E1 -22028.837,E2 -22028.837} C_VEL
LIN {X 0,Y 188.498,Z 626.394,A -85,B 0,C 180,E1 -22029.737,E2 -22029.737} C_VEL
LIN {X 0,Y 187.074,Z 638.123,A -85,B 0,C 180,E1 -22032.228,E2 -22032.228} C_VEL
LIN {X 0,Y 185.933,Z 647.3,A -85,B 0,C 180,E1 -22034.658,E2 -22034.658} C_VEL
LIN {X 0,Y 185.165,Z 655.755,A -85,B 0,C 180,E1 -22037.395,E2 -22037.395} C_VEL
LIN {X 0,Y 184.546,Z 663.954,A -85,B 0,C 180,E1 -22040.686,E2 -22040.686} C_VEL
LIN {X 0,Y 184.466,Z 669.465,A -85,B 0,C 180,E1 -22043.438,E2 -22043.438} C_VEL
LIN {X 0,Y 184.52,Z 674.715,A -85,B 0,C 180,E1 -22046.726,E2 -22046.726} C_VEL
LIN {X 0,Y 184.582,Z 678.625,A -85,B 0,C 180,E1 -22050.001,E2 -22050.001} C_VEL
LIN {X 0,Y 184.221,Z 680.518,A -85,B 0,C 180,E1 -22052.187,E2 -22052.187} C_VEL
LIN {X 0,Y 183.738,Z 682.692,A -85,B 0,C 180,E1 -22056.009,E2 -22056.009} C_VEL
LIN {X 0,Y 183.652,Z 683.473,A -85,B 0,C 180,E1 -22058.806,E2 -22058.806} C_VEL
LIN {X 0,Y 184.506,Z 683.559,A -85,B 0,C 180,E1 -22063.212,E2 -22063.212} C_VEL
LIN {X 0,Y 185.351,Z 683.031,A -85,B 0,C 180,E1 -22065.393,E2 -22065.393} C_VEL
LIN {X 0,Y 188.12,Z 680.891,A -85,B 0,C 180,E1 -22069.648,E2 -22069.648} C_VEL
LIN {X 0,Y 192.245,Z 677.059,A -85,B 0,C 180,E1 -22073.944,E2 -22073.944} C_VEL
LIN {X 0,Y 197.158,Z 672.079,A -85,B 0,C 180,E1 -22077.608,E2 -22077.608} C_VEL
LIN {X 0,Y 201.662,Z 667.034,A -85,B 0,C 180,E1 -22080.354,E2 -22080.354} C_VEL
LIN {X 0,Y 207.848,Z 659.752,A -85,B 0,C 180,E1 -22083.331,E2 -22083.331} C_VEL
LIN {X 0,Y 213.696,Z 652.112,A -85,B 0,C 180,E1 -22085.716,E2 -22085.716} C_VEL
LIN {X 0,Y 220.045,Z 642.937,A -85,B 0,C 180,E1 -22087.94,E2 -22087.94} C_VEL
LIN {X 0,Y 226.372,Z 632.744,A -85,B 0,C 180,E1 -22089.817,E2 -22089.817} C_VEL
LIN {X 0,Y 231.903,Z 622.664,A -85,B 0,C 180,E1 -22091.236,E2 -22091.236} C_VEL
LIN {X 0,Y 237.671,Z 610.568,A -85,B 0,C 180,E1 -22092.566,E2 -22092.566} C_VEL
LIN {X 0,Y 242.703,Z 597.801,A -85,B 0,C 180,E1 -22093.641,E2 -22093.641} C_VEL
LIN {X 0,Y 247.094,Z 584.069,A -85,B 0,C 180,E1 -22094.46,E2 -22094.46} C_VEL
LIN {X 0,Y 250.586,Z 568.707,A -85,B 0,C 180,E1 -22095.171,E2 -22095.171} C_VEL
LIN {X 0,Y 253.524,Z 552.358,A -85,B 0,C 180,E1 -22095.88,E2 -22095.88} C_VEL
LIN {X 0,Y 252.757,Z 547.651,A -85,B 0,C 180,E1 -22097.751,E2 -22097.751} C_VEL
LIN {X 0,Y 252.279,Z 544.169,A -85,B 0,C 180,E1 -22099.633,E2 -22099.633} C_VEL
LIN {X 0,Y 251.961,Z 541.298,A -85,B 0,C 180,E1 -22102.485,E2 -22102.485} C_VEL
LIN {X 0,Y 252.157,Z 540.459,A -85,B 0,C 180,E1 -22104.175,E2 -22104.175} C_VEL
LIN {X 0,Y 253.259,Z 540.692,A -85,B 0,C 180,E1 -22107.375,E2 -22107.375} C_VEL
LIN {X 0,Y 254.381,Z 542.718,A -85,B 0,C 180,E1 -22109.448,E2 -22109.448} C_VEL
LIN {X 0,Y 254.749,Z 543.514,A -85,B 0,C 180,E1 -22110.022,E2 -22110.022} C_VEL
LIN {X 0,Y 250.238,Z 567.013,A -85,B 0,C 180,E1 -22111.073,E2 -22111.073} C_VEL
LIN {X 0,Y 246.69,Z 580.976,A -85,B 0,C 180,E1 -22112.028,E2 -22112.028} C_VEL
LIN {X 0,Y 242.682,Z 592.787,A -85,B 0,C 180,E1 -22113.096,E2 -22113.096} C_VEL
LIN {X 0,Y 238.001,Z 604.027,A -85,B 0,C 180,E1 -22114.414,E2 -22114.414} C_VEL
LIN {X 0,Y 232.637,Z 614.803,A -85,B 0,C 180,E1 -22116.013,E2 -22116.013} C_VEL
LIN {X 0,Y 227.346,Z 623.904,A -85,B 0,C 180,E1 -22117.723,E2 -22117.723} C_VEL
LIN {X 0,Y 221.025,Z 633.281,A -85,B 0,C 180,E1 -22120.012,E2 -22120.012} C_VEL
LIN {X 0,Y 215.156,Z 640.849,A -85,B 0,C 180,E1 -22122.413,E2 -22122.413} C_VEL
LIN {X 0,Y 210.502,Z 646.072,A -85,B 0,C 180,E1 -22124.508,E2 -22124.508} C_VEL
LIN {X 0,Y 203.912,Z 652.528,A -85,B 0,C 180,E1 -22128.065,E2 -22128.065} C_VEL
LIN {X 0,Y 199.211,Z 656.307,A -85,B 0,C 180,E1 -22131.052,E2 -22131.052} C_VEL
LIN {X 0,Y 195.589,Z 658.655,A -85,B 0,C 180,E1 -22133.811,E2 -22133.811} C_VEL
LIN {X 0,Y 193.293,Z 659.845,A -85,B 0,C 180,E1 -22135.83,E2 -22135.83} C_VEL
LIN {X 0,Y 189.458,Z 660.951,A -85,B 0,C 180,E1 -22140,E2 -22140} C_VEL
LIN {X 0,Y 187.904,Z 660.913,A -85,B 0,C 180,E1 -22142.143,E2 -22142.143} C_VEL
LIN {X 0,Y 186.579,Z 660.466,A -85,B 0,C 180,E1 -22144.32,E2 -22144.32} C_VEL
LIN {X 0,Y 184.769,Z 658.432,A -85,B 0,C 180,E1 -22148.518,E2 -22148.518} C_VEL
LIN {X 0,Y 183.838,Z 655.507,A -85,B 0,C 180,E1 -22152.138,E2 -22152.138} C_VEL
LIN {X 0,Y 183.511,Z 651.688,A -85,B 0,C 180,E1 -22155.55,E2 -22155.55} C_VEL
LIN {X 0,Y 183.563,Z 646.648,A -85,B 0,C 180,E1 -22158.992,E2 -22158.992} C_VEL
LIN {X 0,Y 184.03,Z 640.212,A -85,B 0,C 180,E1 -22162.451,E2 -22162.451} C_VEL
LIN {X 0,Y 184.833,Z 632.026,A -85,B 0,C 180,E1 -22165.93,E2 -22165.93} C_VEL
LIN {X 0,Y 185.83,Z 623.626,A -85,B 0,C 180,E1 -22168.829,E2 -22168.829} C_VEL
LIN {X 0,Y 187.08,Z 613.289,A -85,B 0,C 180,E1 -22171.731,E2 -22171.731} C_VEL
LIN {X 0,Y 188.607,Z 601.46,A -85,B 0,C 180,E1 -22174.383,E2 -22174.383} C_VEL
LIN {X 0,Y 190.095,Z 588.819,A -85,B 0,C 180,E1 -22176.595,E2 -22176.595} C_VEL
LIN {X 0,Y 191.333,Z 576.293,A -85,B 0,C 180,E1 -22178.305,E2 -22178.305} C_VEL
LIN {X 0,Y 192.515,Z 562.288,A -85,B 0,C 180,E1 -22179.717,E2 -22179.717} C_VEL
LIN {X 0,Y 193.279,Z 548.948,A -85,B 0,C 180,E1 -22180.659,E2 -22180.659} C_VEL
LIN {X 0,Y 196.245,Z 492.424,A -85,B 0,C 180,E1 -22183.75,E2 -22183.75} C_VEL
LIN {X 0,Y 185.525,Z 460.374,A -85,B 0,C 180,E1 -22186.557,E2 -22186.557} C_VEL
LIN {X 0,Y 185.459,Z 460.383,A -85,B 0,C 180,E1 -22189.892,E2 -22189.892} C_VEL
LIN {X 0,Y 185.502,Z 460.375,A -85,B 0,C 180,E1 -22192.713,E2 -22192.713} C_VEL
LIN {X 0,Y 185.532,Z 460.373,A -85,B 0,C 180,E1 -22197.972,E2 -22197.972} C_VEL
LIN {X 0,Y 185.549,Z 460.371,A -85,B 0,C 180,E1 -22200.594,E2 -22200.594} C_VEL
LIN {X 0,Y 185.582,Z 460.366,A -85,B 0,C 180,E1 -22205.381,E2 -22205.381} C_VEL
LIN {X 0,Y 185.676,Z 460.35,A -85,B 0,C 180,E1 -22211.133,E2 -22211.133} C_VEL
LIN {X 0,Y 185.696,Z 460.355,A -85,B 0,C 180,E1 -22214.637,E2 -22214.637} C_VEL
LIN {X 0,Y 185.889,Z 460.325,A -85,B 0,C 180,E1 -22219.418,E2 -22219.418} C_VEL
LIN {X 0,Y 185.936,Z 460.322,A -85,B 0,C 180,E1 -22223.488,E2 -22223.488} C_VEL
LIN {X 0,Y 186.202,Z 460.288,A -85,B 0,C 180,E1 -22227.836,E2 -22227.836} C_VEL
LIN {X 0,Y 186.4,Z 460.261,A -85,B 0,C 180,E1 -22229.999,E2 -22229.999} C_VEL
LIN {X 0,Y 185.909,Z 460.328,A -85,B 0,C 180,E1 -22234.335,E2 -22234.335} C_VEL
LIN {X 0,Y 185.982,Z 460.316,A -85,B 0,C 180,E1 -22238.693,E2 -22238.693} C_VEL
LIN {X 0,Y 185.724,Z 460.349,A -85,B 0,C 180,E1 -22243.122,E2 -22243.122} C_VEL
LIN {X 0,Y 185.684,Z 460.351,A -85,B 0,C 180,E1 -22247.625,E2 -22247.625} C_VEL
LIN {X 0,Y 185.571,Z 460.37,A -85,B 0,C 180,E1 -22252.254,E2 -22252.254} C_VEL
LIN {X 0,Y 185.577,Z 460.365,A -85,B 0,C 180,E1 -22254.645,E2 -22254.645} C_VEL
LIN {X 0,Y 185.543,Z 460.371,A -85,B 0,C 180,E1 -22259.499,E2 -22259.499} C_VEL
LIN {X 0,Y 185.496,Z 460.375,A -85,B 0,C 180,E1 -22264.632,E2 -22264.632} C_VEL
LIN {X 0,Y 185.5,Z 460.377,A -85,B 0,C 180,E1 -22267.314,E2 -22267.314} C_VEL
LIN {X 0,Y 185.462,Z 460.381,A -85,B 0,C 180,E1 -22270.722,E2 -22270.722} C_VEL
LIN {X 0,Y 185.457,Z 460.382,A -85,B 0,C 180,E1 -22276.055,E2 -22276.055} C_VEL
LIN {X 0,Y 185.466,Z 460.38,A -85,B 0,C 180,E1 -22279.895,E2 -22279.895} C_VEL
LIN {X 0,Y 185.505,Z 460.376,A -85,B 0,C 180,E1 -22282.711,E2 -22282.711} C_VEL
LIN {X 0,Y 185.541,Z 460.371,A -85,B 0,C 180,E1 -22287.974,E2 -22287.974} C_VEL
LIN {X 0,Y 185.579,Z 460.365,A -85,B 0,C 180,E1 -22290.576,E2 -22290.576} C_VEL
LIN {X 0,Y 185.587,Z 460.366,A -85,B 0,C 180,E1 -22295.382,E2 -22295.382} C_VEL
LIN {X 0,Y 185.693,Z 460.353,A -85,B 0,C 180,E1 -22301.115,E2 -22301.115} C_VEL
LIN {X 0,Y 185.722,Z 460.351,A -85,B 0,C 180,E1 -22304.64,E2 -22304.64} C_VEL
LIN {X 0,Y 185.923,Z 460.323,A -85,B 0,C 180,E1 -22309.359,E2 -22309.359} C_VEL
LIN {X 0,Y 185.962,Z 460.319,A -85,B 0,C 180,E1 -22313.49,E2 -22313.49} C_VEL
LIN {X 0,Y 186.206,Z 460.286,A -85,B 0,C 180,E1 -22317.837,E2 -22317.837} C_VEL
LIN {X 0,Y 186.406,Z 460.264,A -85,B 0,C 180,E1 -22320,E2 -22320} C_VEL
LIN {X 0,Y 185.926,Z 460.323,A -85,B 0,C 180,E1 -22324.336,E2 -22324.336} C_VEL
LIN {X 0,Y 186.024,Z 460.314,A -85,B 0,C 180,E1 -22328.692,E2 -22328.692} C_VEL
LIN {X 0,Y 185.764,Z 460.34,A -85,B 0,C 180,E1 -22333.121,E2 -22333.121} C_VEL
LIN {X 0,Y 185.674,Z 460.357,A -85,B 0,C 180,E1 -22338.867,E2 -22338.867} C_VEL
LIN {X 0,Y 185.576,Z 460.368,A -85,B 0,C 180,E1 -22344.646,E2 -22344.646} C_VEL
LIN {X 0,Y 185.578,Z 460.365,A -85,B 0,C 180,E1 -22349.493,E2 -22349.493} C_VEL
LIN {X 0,Y 185.499,Z 460.379,A -85,B 0,C 180,E1 -22354.632,E2 -22354.632} C_VEL
LIN {X 0,Y 185.505,Z 460.376,A -85,B 0,C 180,E1 -22357.314,E2 -22357.314} C_VEL
LIN {X 0,Y 185.471,Z 460.378,A -85,B 0,C 180,E1 -22360.726,E2 -22360.726} C_VEL
LIN {X 0,Y 185.461,Z 460.381,A -85,B 0,C 180,E1 -22366.055,E2 -22366.055} C_VEL
